(* IEC 61131-3 sources: xPLCCore/codesys_code/Application/APPs, 7 files *)

(* ---- AxisGroupSM.st ---- *)
PROGRAM AxisGroupSM
    VAR CONSTANT
        FlyEventBufferSize: UDINT := 10;
        TaskInstructionBufferSize: UDINT := 10;
        FlyEventStageLimit: INT := 9;

        // Motion buffer fullness threshold: reject new 'M' packets when the
        // SoftMotion command buffer has this many queued moves (back-pressure).
        MOTION_BUFFER_THRESHOLD : ULINT := 12;
        // Cooldown (ms) before re-trying a motion command after the FB
        // refused .CommandAccepted (e.g. GroupWait, MoveLinearAbsolute).
        RETRY_COOLDOWN_G4_MS    : DINT := 100;
        RETRY_COOLDOWN_G1_MS    : DINT := 101;
        // Error code reported on FlyEvent TimeToLive expiry.
        TRIGGER_TIMEOUT_ERR     : INT := 100;
        // Sentinel used by 'G1' to detect "A not supplied" in the TryReadREAL
        // default. Any real A value is << |919191|.
        G1_A_UNSET_SENTINEL     : LREAL := -919191;
    END_VAR
    VAR
        reelpullmotor_fActPosition:REAL;
		OutputCHs:ARRAY[0..15] OF USINT;
		InputCHs:ARRAY[0..15] OF USINT;
		RuntimeMs: LINT := 0;
        BusPeriod: DINT := 1;
        AxisGroupReady: BOOL := FALSE;

        AxisGroupManagerFb: AxisGroupManager(
            agAxisGroup := AxisGroupGVL_agSpiderR.SpiderR,
			axReel:=reelpullmotor);

        GroupActualPositionFb: SM3_Robotics.MC_GroupReadActualPosition;
        ReadPosition: SM3_Robotics.SMC_POS_REF;

        SetCoordTransformFb : MC_SetCoordinateTransform;
        ReadMcsTransformFb : MC_ReadCoordinateTransform;
        ApplyCoordTransform : BOOL := FALSE;
        CoordTransform : MC_COORD_REF;

        InputEvent: E_RobotEvent := E_RobotEvent.EV_NONE;
        PreviousInputEvent: E_RobotEvent := E_RobotEvent.EV_NONE;
        VisuEventControl: INT;
        StateString: STRING;

        MotionStateString: STRING;

        reelMoveRelative : MC_MoveRelative;
        reelMoveRelative2: MC_MoveRelative;   // second instance: SoftMotion forbids >1 movement per FB
        // Request-pattern vars for cyclic reelMoveRelative
        reelGoRequest  : BOOL  := FALSE;
        reelGoRequest2 : BOOL  := FALSE;
        reelGoDistance : LREAL := 0;
        reelGoVelocity : LREAL := 0;
        reelGoAccel    : LREAL := 100;
        reelGoDecel    : LREAL := 100;
        reelGoJerk     : LREAL := 1000;

        MoveLinearAbsoluteFb: SM3_Robotics.MC_MoveLinearAbsolute;
        GroupWaitFb: SM3_Robotics.SMC_GroupWait;

        MotionPose: SM3_Robotics.SMC_POS_REF := ( c := (x := 0.0, y := 0.0, z := 0.0, a := 0.0));

        PacketType: STRING;
        CommandType: STRING;
        CommandId: DINT := 0;
        ShouldReturn: BOOL := FALSE;
        CommandAck: BOOL := FALSE;

        MessageUnpackerFb: FB_MpUnpacker;
        fbPinOpSeqUnpacker: FB_MpUnpacker; // Helper unpacker for pin_op_seq array

        FlyEventBuffer: ARRAY [0..FlyEventBufferSize-1] OF FlyEventData; // event queue for motion-triggered IO
        FlyEventAvailableCount: INT;

        // TaskInstructionBuffer: ARRAY [0..TaskInstructionBufferSize-1] OF TaskInstructionData;
        // TaskInstructionBuffer_ridx:FB_RingBufferIndex(TaskInstructionBufferSize);

        RetryMotionCommandCooldown: DINT := 0;

        LatestFeedRate: LREAL := 10000;
        LatestAcceleration: LREAL := 10000;
        LatestDeceleration: LREAL := 10000;
        LatestJerk: LREAL := 10000;
        LatestFactor: LREAL := 1;

        CornerTransition: REAL := 3;

        GroupReadStatusFb: SM3_Robotics.MC_GroupReadStatus;
        GroupReadPositionFb: SM3_Robotics.SMC_GroupReadPositionInMovement;
        GroupReadPositionFb2: SM3_Robotics.SMC_GroupReadPositionInMovement;

        MotionBufferSize: ULINT;
        CurrentMovementId: SMC_Movement_Id;
        CurrentMovementIdProgress: REAL;

        MessagePackerFb: FB_MpPacker;
        ResponsePacketPointer: POINTER TO MsgPakInfo;

        // MaxVelocity: REAL := 1000;
        // MaxAcceleration: REAL := 4000;
        // MaxJerk: REAL := 4000000;

        DigitalOutputBits: ULINT;
        TmpDigitalOutputBits: ULINT;

        IoTriggerCount: INT := 0;
        IoTriggerResetCount: INT := 0;
        IoTriggerInfoCount: INT := 0;
        IoCommandCount: INT := 0;

        DigitalInputBits_Curr: ULINT := 0;
        DigitalInputBits_Prev: ULINT := 0;
        DigitalInputFlipCounts: ARRAY[0..15] OF UDINT;

        PrevAxisGroupState: INT := -1; // Force initial StateString update

    Index : INT;
    StageLoopIdx : INT;
    PinOpSeqIdx : INT; // Index for iterating through pin_op_seq array

    TempMovementId : SMC_Movement_Id;

    MessageBufferPointer : POINTER TO BYTE;
    AuxCommandBufferPointer : POINTER TO BYTE;

    TriggerActive : BOOL;
    TriggerErrorCode : INT;
    TempByte : BYTE;
    DigitalOutputPointer : POINTER TO BYTE;

        MotionOutputPin: ULINT;
        StagePinState: ULINT;
        StagePinMaskTemp: ULINT;
        StagePinStateTemp: ULINT;
        StageDelayTemp: DINT;

    //LocVar FOR ProcessMotionPacket
    TransitionParameter : ARRAY [0..1] OF LREAL := [0, 0];
    FlyEventTempData : FlyEventData;
    MotionPoseTempReal : REAL;
    PrevMotionStateId : SMC_Movement_Id; // For MotionStateString change detection
    PrevMotionStateProgress : REAL := -1.0; // Force initial update
    G1AbortMode : BOOL; // TRUE = BufferMode.Aborting, interrupts current move

    G4HaltTime: REAL;
    InputPinMask: UINT;
    InputPinGroup: UINT;
    InputPinState: UINT;

    MotionTargetMovementId: SMC_Movement_Id;

    DigitalInputPointer: POINTER TO BYTE;

    DBG_PIN: UINT;

    DBG_BLOCK : BOOL:=TRUE;

    END_VAR
(* =========== IMPLEMENTATION =========== *)

//IMPORTANT:following if TRUE... and if FALSE.... are mandatory, DO not try to remove/optimize it

    //InitRuntime();
    IF TRUE THEN
        IF RuntimeMs = 0 THEN
            FOR Index := 0 TO GVL.reMP_info_ridx.capacity() - 1 DO
                GVL.reMP_info_arr[Index] := MsgPakInfoInit(
                    buff := ADR(GVL.reMP_info_buf[Index]),
                    buffer_size := GVL.reMP_info_buff_SIZE,
                    useLargeElementCountField := TRUE
                );
            END_FOR
        END_IF;
    END_IF;

    // Virtual-motors TTL gate. Derive GVL.bVirtualMotorsMode from
    // GVL.bVirtualMotorsMode_Request (which the operator forces via
    // CODESYS online mode) and a self-expiring timer. Even if the force
    // is left on indefinitely, the derived flag snaps back to FALSE
    // after VIRTUAL_MOTORS_TTL so a forgotten override can't leak into
    // a real-motor session without a cold boot. See GVL.st for docs.
    GVL.fbVirtualMotorsExpire(IN := GVL.bVirtualMotorsMode_Request, PT := GVL.VIRTUAL_MOTORS_TTL);
    GVL.bVirtualMotorsMode := GVL.bVirtualMotorsMode_Request AND NOT GVL.fbVirtualMotorsExpire.Q;

    //UpdateRuntimeAndInputEvent();
    IF TRUE THEN
        RuntimeMs := RuntimeMs + BusPeriod;

        // VisuEventControl=0 is the idle/no-op default so the TCP handler
        // (ProcessSystemPacket below) can own InputEvent without being
        // clobbered by this block on the next cycle. Visualisation buttons
        // should write 1..6 momentarily and reset to 0.
        CASE VisuEventControl OF
            1: InputEvent := E_RobotEvent.EV_POWER_ON;
            2: InputEvent := E_RobotEvent.EV_GROUP_ENABLE;
            3: InputEvent := E_RobotEvent.EV_HOME_GO;
            4: InputEvent := E_RobotEvent.EV_ERROR;
            5: InputEvent := E_RobotEvent.EV_RESET;
            6: InputEvent := E_RobotEvent.EV_HOME_GO_FORCE_SKIP;
        END_CASE;

        IF (PreviousInputEvent <> InputEvent) THEN
            AxisGroupManagerFb.TRANSITION(
                eEvent := InputEvent
            );
        END_IF;

        PreviousInputEvent := InputEvent;
        IF TO_INT(AxisGroupManagerFb._eState) <> PrevAxisGroupState THEN
            StateString := TO_STRING(AxisGroupManagerFb._eState);
            PrevAxisGroupState := TO_INT(AxisGroupManagerFb._eState);
        END_IF;
    END_IF;

    //UpdateAxisGroupState();
    IF TRUE THEN
        AxisGroupManagerFb.Update();

        GroupReadStatusFb(
            AxisGroup := AxisGroupManagerFb._agAxisGroup,
            Enable := 1,
            ActiveMovementId =>
        );

        GroupReadPositionFb(
            AxisGroup := AxisGroupManagerFb._agAxisGroup,
            Enable := TRUE
        );

        GroupActualPositionFb(
            AxisGroup := AxisGroupManagerFb._agAxisGroup,
            Enable := 1,
            CoordSystem := SMC_COORD_SYSTEM.WCS,
            Position => ReadPosition,
        );

    END_IF;

    // Global error supervisor: the per-state checks in AxisGroupManager.Update
    // only watch the power FBs. A move that goes into errorstop (axis fault,
    // bus drop mid-motion, servo trip) surfaces on GroupReadStatusFb.Error /
    // GroupReadPositionFb.Error, and a bus-level fault on
    // IoConfig_Globals.EtherCAT_Master_SoftMotion.xError. Catch those here
    // and drive the FSM to Error -- guarded so we don't loop while already
    // in Error/UnInited. Bus errors take priority so the error source is
    // diagnostic rather than a downstream symptom.
    IF (AxisGroupManagerFb._eState <> E_RobotState.Error
        AND AxisGroupManagerFb._eState <> E_RobotState.UnInited) THEN
        IF IoConfig_Globals.EtherCAT_Master_SoftMotion.xError THEN
            GVL.LastErrorSource := 'Supervisor:EtherCAT_Master';
            GVL.LastErrorID := 0;
            AxisGroupManagerFb.Transition(E_RobotEvent.EV_ERROR);
        ELSIF GroupReadStatusFb.Error THEN
            GVL.LastErrorSource := 'Supervisor:GroupReadStatus';
            GVL.LastErrorID := TO_DWORD(GroupReadStatusFb.ErrorID);
            AxisGroupManagerFb.Transition(E_RobotEvent.EV_ERROR);
        ELSIF GroupReadPositionFb.Error THEN
            GVL.LastErrorSource := 'Supervisor:GroupReadPosition';
            GVL.LastErrorID := TO_DWORD(GroupReadPositionFb.ErrorID);
            AxisGroupManagerFb.Transition(E_RobotEvent.EV_ERROR);
        END_IF;
    END_IF;

    //UpdateMotionProgress();
    IF TRUE THEN
        TempMovementId := GroupReadPositionFb.MovementId;
        // If either MC read FB is in error, don't propagate its outputs -- they
        // may be stale. Freeze buffer size to 0 so ProcessMotionPacket won't
        // treat "buffer has room" as "motion is healthy" and accept a new
        // move on top of an errored group.
        IF GroupReadStatusFb.Error OR GroupReadPositionFb.Error THEN
            MotionBufferSize := 0;
        ELSIF (GroupReadPositionFb.MovementId = 0) THEN
            MotionBufferSize := 0;
            CurrentMovementId := GroupReadStatusFb.LastAcceptedMovementId;
            CurrentMovementIdProgress := 1;
            IF (CurrentMovementId = 0) THEN
                CurrentMovementIdProgress := 0;
            END_IF;
        ELSE
            // Guard against underflow: both are unsigned SMC_Movement_Id.
            // LastAccepted < current shouldn't happen, but could during
            // a reset race. Clamp to 0 rather than wrapping to huge ULINT.
            IF GroupReadStatusFb.LastAcceptedMovementId >= GroupReadPositionFb.MovementId THEN
                MotionBufferSize := GroupReadStatusFb.LastAcceptedMovementId - GroupReadPositionFb.MovementId;
            ELSE
                MotionBufferSize := 0;
            END_IF;

            IF (CurrentMovementId <> GroupReadPositionFb.MovementId) THEN
                CurrentMovementId := GroupReadPositionFb.MovementId;
            END_IF;

            CurrentMovementIdProgress := GroupReadPositionFb.Position;
        END_IF;

        IF (CurrentMovementId <> PrevMotionStateId OR CurrentMovementIdProgress <> PrevMotionStateProgress) THEN
            MotionStateString := CONCAT(
                CONCAT(TO_STRING(CurrentMovementId), ' '),
                TO_STRING(CurrentMovementIdProgress)
            );
            PrevMotionStateId := CurrentMovementId;
            PrevMotionStateProgress := CurrentMovementIdProgress;
        END_IF;

        ShouldReturn := FALSE;
        CommandAck := FALSE;

    END_IF;

    //ReadIncomingPacket();
    IF TRUE THEN
        PacketType := '';
        ResponsePacketPointer := 0;

        IF (GVL.minfo_buf_ridx.size() > 0) THEN
            MessageBufferPointer := ADR(GVL.minfo_buf[GVL.minfo_buf_ridx.getTail()][0]);
            MessageUnpackerFb.Init(ADR(MessageBufferPointer[1]), MessageBufferPointer[0]);
            CommandId := TO_DINT(MessageUnpackerFb.TryReadINT64('id', - 1));
            PacketType := MessageUnpackerFb.TryReadString('type', '');
            CommandType := MessageUnpackerFb.TryReadString('cmd', '');
        END_IF;
    END_IF;

    IF TRUE THEN//ProcessSystemPacket

        IF (PacketType = 'SYS') THEN
            // reMP overflow guard: if the reply ring is full, drop the oldest
            // queued reply to make room. getHead() returning -1 would index
            // reMP_info_arr[-1] and fault the task. See doc/ringbuf-bugs.md #4.
            IF (GVL.reMP_info_ridx.space() = 0) THEN
                GVL.reMP_info_ridx.consumeTail();
                GVL.ReMpDropCount := GVL.ReMpDropCount + 1;
            END_IF;
            ResponsePacketPointer := ADR(GVL.reMP_info_arr[GVL.reMP_info_ridx.getHead()]); // prepare for return data buffer

            MsgPakInfoClear(ResponsePacketPointer^);

            IF (CommandType = 'GA_EV') THEN
                ShouldReturn := TRUE;
                CommandAck := TRUE;
                InputEvent := TO_UDINT(MessageUnpackerFb.TryReadINT64('ev', - 1));
                AxisGroupManagerFb.TRANSITION(
                    eEvent := InputEvent
                );

                ShouldReturn := TRUE;
                CommandAck := TRUE;
                ResponsePacketPointer^.ele_count := 4;
                ResponsePacketPointer^.whead := MessagePackerFb.PackString(pStart := ResponsePacketPointer^.whead, psValue := ADR('st'));
                ResponsePacketPointer^.whead := MessagePackerFb.PackDINT(pStart := ResponsePacketPointer^.whead, diValue := AxisGroupManagerFb._eState);
                ResponsePacketPointer^.whead := MessagePackerFb.PackString(pStart := ResponsePacketPointer^.whead, psValue := ADR('st_str'));
                StateString := TO_STRING(AxisGroupManagerFb._eState);
                PrevAxisGroupState := TO_INT(AxisGroupManagerFb._eState);
                ResponsePacketPointer^.whead := MessagePackerFb.PackString(pStart := ResponsePacketPointer^.whead, psValue := ADR(StateString));
                // Error latch: empty string + 0 when no error has been recorded
                // since the last EV_RESET -> UnInited cycle.
                ResponsePacketPointer^.whead := MessagePackerFb.PackString(pStart := ResponsePacketPointer^.whead, psValue := ADR('err_src'));
                ResponsePacketPointer^.whead := MessagePackerFb.PackString(pStart := ResponsePacketPointer^.whead, psValue := ADR(GVL.LastErrorSource));
                ResponsePacketPointer^.whead := MessagePackerFb.PackString(pStart := ResponsePacketPointer^.whead, psValue := ADR('err_id'));
                ResponsePacketPointer^.whead := MessagePackerFb.PackDINT(pStart := ResponsePacketPointer^.whead, diValue := TO_DINT(GVL.LastErrorID));
            ELSE
                // Unknown SYS command -- emit NAK so the TS caller doesn't hang on timeout.
                ShouldReturn := TRUE;
                CommandAck := FALSE;
                ResponsePacketPointer^.ele_count := 1;
                ResponsePacketPointer^.whead := MessagePackerFb.PackString(pStart := ResponsePacketPointer^.whead, psValue := ADR('err'));
                ResponsePacketPointer^.whead := MessagePackerFb.PackString(pStart := ResponsePacketPointer^.whead, psValue := ADR('unknown SYS cmd'));
            END_IF;

            GVL.minfo_buf_ridx.consumeTail();

            IF ShouldReturn = TRUE THEN // return ack/nak with id
                ResponsePacketPointer^.whead := MessagePackerFb.PackString(pStart := ResponsePacketPointer^.whead, psValue := ADR('id'));
                ResponsePacketPointer^.whead := MessagePackerFb.PackDINT(pStart := ResponsePacketPointer^.whead, diValue := CommandId);

                ResponsePacketPointer^.whead := MessagePackerFb.PackString(pStart := ResponsePacketPointer^.whead, psValue := ADR('ack'));
                ResponsePacketPointer^.whead := MessagePackerFb.PackBool(pStart := ResponsePacketPointer^.whead, bValue := CommandAck);

                ResponsePacketPointer^.ele_count := ResponsePacketPointer^.ele_count + 2;
                MsgPakInfoWrapup(ResponsePacketPointer^);
                GVL.reMP_info_ridx.pushHead();
            END_IF;
        END_IF;

    END_IF;

    IF TRUE THEN//ProcessAuxCommands
        // AUX command threads: currently drained without parsing so their ring
        // buffers don't back up and block the client. Wire a real handler here
        // when the AUX command feature is implemented (see README §P2 #10).
        IF (GVL.aux0_info_buf_ridx.size() > 0) THEN
            AuxCommandBufferPointer := ADR(GVL.aux0_info_buf[GVL.aux0_info_buf_ridx.getTail()][0]);
            GVL.aux0_info_buf_ridx.consumeTail();
        END_IF;

        IF (GVL.aux1_info_buf_ridx.size() > 0) THEN
            AuxCommandBufferPointer := ADR(GVL.aux1_info_buf[GVL.aux1_info_buf_ridx.getTail()][0]);
            GVL.aux1_info_buf_ridx.consumeTail();
        END_IF;

        IF (GVL.aux2_info_buf_ridx.size() > 0) THEN
            AuxCommandBufferPointer := ADR(GVL.aux2_info_buf[GVL.aux2_info_buf_ridx.getTail()][0]);
            GVL.aux2_info_buf_ridx.consumeTail();
        END_IF;
    END_IF;

   //OutputCHs[1]:=InputCHs[1];
   //OutputCHs[2]:=InputCHs[2];
   //OutputCHs[3]:=InputCHs[2];

   // DigitalInputPointer := IoConfig_Globals.HECAT_1616.InputData;//////////////////////////////////////////////

    IF DigitalInputPointer <> 0 THEN//TrackDigitalInputFlips
        DigitalInputBits_Curr := TO_ULINT(DigitalInputPointer[0]) OR SHL(TO_ULINT(DigitalInputPointer[1]), 8);
        IF RuntimeMs > 1 THEN
            TmpDigitalOutputBits := DigitalInputBits_Curr XOR DigitalInputBits_Prev;
            IF TmpDigitalOutputBits <> 0 THEN
                FOR Index := 0 TO 15 DO
                    IF (SHR(TmpDigitalOutputBits, TO_DINT(Index)) AND 1) <> 0 THEN
                        DigitalInputFlipCounts[Index] := DigitalInputFlipCounts[Index] + 1;
                    END_IF;
                END_FOR;
            END_IF;
        END_IF;
        DigitalInputBits_Prev := DigitalInputBits_Curr;
    END_IF;

    IF TRUE THEN//CheckAxisGroupReady
        AxisGroupReady := (AxisGroupManagerFb._eState = E_RobotState.Ready);

        IF NOT AxisGroupReady THEN
            // Host-authority gate (solidification.md W1 A1). Previously this
            // block called GVL.minfo_buf_ridx.clear() which silently dropped
            // every queued motion packet with no reply -- the UI's
            // sendTcpMsgPack would hang until its own timeout. Drain each
            // packet with an explicit NAK + err='group_not_ready' so the
            // host can distinguish "PLC not ready" from "PLC dead".
            // SYS/AUX paths above already ran and are unaffected.
            WHILE GVL.minfo_buf_ridx.size() > 0 DO
                // Re-parse each slot's header to get CommandId for the echo.
                MessageBufferPointer := ADR(GVL.minfo_buf[GVL.minfo_buf_ridx.getTail()][0]);
                MessageUnpackerFb.Init(ADR(MessageBufferPointer[1]), MessageBufferPointer[0]);
                CommandId := TO_DINT(MessageUnpackerFb.TryReadINT64('id', -1));

                // reMP overflow guard (see doc/ringbuf-bugs.md #4).
                IF (GVL.reMP_info_ridx.space() = 0) THEN
                    GVL.reMP_info_ridx.consumeTail();
                    GVL.ReMpDropCount := GVL.ReMpDropCount + 1;
                END_IF;
                ResponsePacketPointer := ADR(GVL.reMP_info_arr[GVL.reMP_info_ridx.getHead()]);
                MsgPakInfoClear(ResponsePacketPointer^);
                ResponsePacketPointer^.ele_count := ResponsePacketPointer^.ele_count + 3;
                ResponsePacketPointer^.whead := MessagePackerFb.PackString(pStart := ResponsePacketPointer^.whead, psValue := ADR('err'));
                ResponsePacketPointer^.whead := MessagePackerFb.PackString(pStart := ResponsePacketPointer^.whead, psValue := ADR('group_not_ready'));
                ResponsePacketPointer^.whead := MessagePackerFb.PackString(pStart := ResponsePacketPointer^.whead, psValue := ADR('id'));
                ResponsePacketPointer^.whead := MessagePackerFb.PackDINT(pStart := ResponsePacketPointer^.whead, diValue := CommandId);
                ResponsePacketPointer^.whead := MessagePackerFb.PackString(pStart := ResponsePacketPointer^.whead, psValue := ADR('ack'));
                ResponsePacketPointer^.whead := MessagePackerFb.PackBool(pStart := ResponsePacketPointer^.whead, bValue := FALSE);
                MsgPakInfoWrapup(ResponsePacketPointer^);
                GVL.reMP_info_ridx.pushHead();

                GVL.minfo_buf_ridx.consumeTail();
                GVL.GroupNotReadyNakCount := GVL.GroupNotReadyNakCount + 1;
            END_WHILE;

            MotionPose.c.X := 0;
            MotionPose.c.Y := 0;
            MotionPose.c.Z := 0;
            MotionPose.c.A := 0;
            MotionPose.c.B := 0;
            MotionPose.c.C := 0;
        END_IF;
    END_IF;

    IF NOT AxisGroupReady THEN
        RETURN;
    END_IF;

    IF FALSE THEN///ProcessTaskPacket

        IF (PacketType = 'TASK') THEN
            ResponsePacketPointer := ADR(GVL.reMP_info_arr[GVL.reMP_info_ridx.getHead()]); // prepare for return data buffer

            MsgPakInfoClear(ResponsePacketPointer^);

            IF (CommandType = 'GA_EV') THEN
            	Index:=0;
            END_IF;

            GVL.minfo_buf_ridx.consumeTail();

            IF ShouldReturn = TRUE THEN // return ack/nak with id
                ResponsePacketPointer^.whead := MessagePackerFb.PackString(pStart := ResponsePacketPointer^.whead, psValue := ADR('id'));
                ResponsePacketPointer^.whead := MessagePackerFb.PackDINT(pStart := ResponsePacketPointer^.whead, diValue := CommandId);

                ResponsePacketPointer^.whead := MessagePackerFb.PackString(pStart := ResponsePacketPointer^.whead, psValue := ADR('ack'));
                ResponsePacketPointer^.whead := MessagePackerFb.PackBool(pStart := ResponsePacketPointer^.whead, bValue := CommandAck);

                ResponsePacketPointer^.ele_count := ResponsePacketPointer^.ele_count + 2;
                MsgPakInfoWrapup(ResponsePacketPointer^);
                GVL.reMP_info_ridx.pushHead();
            END_IF;
        END_IF;

    END_IF;

    IF TRUE THEN//ProcessFlyEventsAndIo

        TriggerActive := FALSE;
        FlyEventAvailableCount := 0;

        FOR Index := 0 TO TO_INT(FlyEventBufferSize - 1) DO
            TriggerActive := FALSE;
            TriggerErrorCode := 0;

            CASE FlyEventBuffer[Index].TriggerType OF
                FlyEventTriggerType.MovmentProgressTrigger:
                    IF (
                        CurrentMovementId > FlyEventBuffer[Index].TargetMovementId OR
                        (CurrentMovementId = FlyEventBuffer[Index].TargetMovementId AND CurrentMovementIdProgress >= FlyEventBuffer[Index].TargetMovementProgress)
                    ) THEN
                        TriggerActive := TRUE;
                        IF (FlyEventBuffer[Index].IoStageCount > 0) THEN
                            FlyEventBuffer[Index].IoStageIndex := 0;
                            FlyEventBuffer[Index].IoStageDelayCountdown := FlyEventBuffer[Index].IoStageDelay[0];
                            FlyEventBuffer[Index].TriggerType := FlyEventTriggerType.SequenceDelayWait;
                            IF (FlyEventBuffer[Index].IoStageDelayCountdown > 0) THEN
                                TriggerActive := FALSE;
                            END_IF;
                        END_IF;
                    ELSE
                        IF (FlyEventBuffer[Index].TimeToLiveMs > 0) THEN
                            FlyEventBuffer[Index].TimeToLiveMs := FlyEventBuffer[Index].TimeToLiveMs - BusPeriod;
                            IF (FlyEventBuffer[Index].TimeToLiveMs <= 0) THEN
                                TriggerActive := TRUE;
                                TriggerErrorCode := TRIGGER_TIMEOUT_ERR;
                            END_IF;
                        END_IF;
                    END_IF;

                FlyEventTriggerType.SequenceDelayWait:
                    IF (FlyEventBuffer[Index].IoStageIndex < FlyEventBuffer[Index].IoStageCount) THEN
                        FlyEventBuffer[Index].IoStageDelayCountdown := FlyEventBuffer[Index].IoStageDelayCountdown - BusPeriod;
                        IF (FlyEventBuffer[Index].IoStageDelayCountdown <= 0) THEN
                            TriggerActive := TRUE;
                        END_IF;
                    END_IF;

                FlyEventTriggerType.NOP:
                    FlyEventAvailableCount := FlyEventAvailableCount + 1;
            END_CASE;

            IF (TriggerActive = FALSE) THEN
                CONTINUE;
            END_IF;

            IF (TriggerErrorCode <> 0) THEN
                // reMP overflow guard (see doc/ringbuf-bugs.md #4).
                IF (GVL.reMP_info_ridx.space() = 0) THEN
                    GVL.reMP_info_ridx.consumeTail();
                    GVL.ReMpDropCount := GVL.ReMpDropCount + 1;
                END_IF;
                ResponsePacketPointer := ADR(GVL.reMP_info_arr[GVL.reMP_info_ridx.getHead()]); // prepare for return data buffer
                MsgPakInfoClear(ResponsePacketPointer^);
                ResponsePacketPointer^.ele_count := ResponsePacketPointer^.ele_count + 3;

                ResponsePacketPointer^.whead := MessagePackerFb.PackString(pStart := ResponsePacketPointer^.whead, psValue := ADR('error_code'));
                ResponsePacketPointer^.whead := MessagePackerFb.PackDINT(pStart := ResponsePacketPointer^.whead, diValue := TriggerErrorCode);

                ResponsePacketPointer^.whead := MessagePackerFb.PackString(pStart := ResponsePacketPointer^.whead, psValue := ADR('src_id'));
                ResponsePacketPointer^.whead := MessagePackerFb.PackDINT(pStart := ResponsePacketPointer^.whead, diValue := FlyEventBuffer[Index].SourceCommandId);

                ResponsePacketPointer^.whead := MessagePackerFb.PackString(pStart := ResponsePacketPointer^.whead, psValue := ADR('event_id'));
                ResponsePacketPointer^.whead := MessagePackerFb.PackLINT(pStart := ResponsePacketPointer^.whead, liValue := TO_LINT(FlyEventBuffer[Index].EventId));

                MsgPakInfoWrapup(ResponsePacketPointer^);
                GVL.reMP_info_ridx.pushHead();

                FlyEventBuffer[Index].ActionType := FlyEventActType.NOP;
                FlyEventBuffer[Index].TriggerType := FlyEventTriggerType.NOP;
            ELSE
                CASE FlyEventBuffer[Index].ActionType OF
                    FlyEventActType.PIN_OPERATION:
                        IF (FlyEventBuffer[Index].IoStageCount > 0) THEN
                            MotionOutputPin := FlyEventBuffer[Index].IoStagePinMask[FlyEventBuffer[Index].IoStageIndex];
                            StagePinState := FlyEventBuffer[Index].IoStagePinState[FlyEventBuffer[Index].IoStageIndex];
                        ELSE
                            MotionOutputPin := 0;
                            StagePinState := 0;
                        END_IF;

                        TmpDigitalOutputBits := DigitalOutputBits;
                        TmpDigitalOutputBits :=
                            (TmpDigitalOutputBits AND NOT (MotionOutputPin)) OR
                            ((StagePinState) AND (MotionOutputPin));
                        DigitalOutputBits := TmpDigitalOutputBits;

                        FlyEventBuffer[Index].IoStageIndex := FlyEventBuffer[Index].IoStageIndex + 1;
                        IF (FlyEventBuffer[Index].IoStageIndex < FlyEventBuffer[Index].IoStageCount) THEN
                            FlyEventBuffer[Index].IoStageDelayCountdown := FlyEventBuffer[Index].IoStageDelay[FlyEventBuffer[Index].IoStageIndex];
                            FlyEventBuffer[Index].TriggerType := FlyEventTriggerType.SequenceDelayWait;
                        ELSE
                            FlyEventBuffer[Index].ActionType := FlyEventActType.NOP;
                            FlyEventBuffer[Index].TriggerType := FlyEventTriggerType.NOP;
                        END_IF;

                        IoTriggerCount := IoTriggerCount + 1;

                    FlyEventActType.ACK_SRC_ID://send ack with source command id
                        // reMP overflow guard (see doc/ringbuf-bugs.md #4).
                        IF (GVL.reMP_info_ridx.space() = 0) THEN
                            GVL.reMP_info_ridx.consumeTail();
                            GVL.ReMpDropCount := GVL.ReMpDropCount + 1;
                        END_IF;

                        ResponsePacketPointer := ADR(GVL.reMP_info_arr[GVL.reMP_info_ridx.getHead()]); // prepare for return data buffer
                        MsgPakInfoClear(ResponsePacketPointer^);

                        ResponsePacketPointer^.ele_count := ResponsePacketPointer^.ele_count +3;//three elements: event_id, id, ack

                        ResponsePacketPointer^.whead := MessagePackerFb.PackString(pStart := ResponsePacketPointer^.whead, psValue := ADR('event_id'));
                        ResponsePacketPointer^.whead := MessagePackerFb.PackLINT(pStart := ResponsePacketPointer^.whead, liValue := TO_LINT(FlyEventBuffer[Index].EventId));

                        ResponsePacketPointer^.whead := MessagePackerFb.PackString(pStart := ResponsePacketPointer^.whead, psValue := ADR('id'));
                        ResponsePacketPointer^.whead := MessagePackerFb.PackDINT(pStart := ResponsePacketPointer^.whead, diValue := FlyEventBuffer[Index].SourceCommandId);

                        ResponsePacketPointer^.whead := MessagePackerFb.PackString(pStart := ResponsePacketPointer^.whead, psValue := ADR('ack'));
                        ResponsePacketPointer^.whead := MessagePackerFb.PackBool(pStart := ResponsePacketPointer^.whead, bValue := TRUE);

                        MsgPakInfoWrapup(ResponsePacketPointer^);
                        GVL.reMP_info_ridx.pushHead();

                        // IF (FlyEventBuffer[Index].SourceCommandId = CommandId) THEN
                        //     TriggerActive := TRUE;
                        // END_IF;

                        FlyEventBuffer[Index].ActionType := FlyEventActType.NOP;
                        FlyEventBuffer[Index].TriggerType := FlyEventTriggerType.NOP;

                END_CASE;
            END_IF;

            IoTriggerInfoCount := IoTriggerInfoCount + 1;
        END_FOR;

        //DigitalOutputPointer := IoConfig_Globals.HECAT_1616.OutputData;//////////////////////////////////////////////
        OutputCHs[0] := TO_BYTE(DigitalOutputBits AND 16#FF);
        OutputCHs[1] := TO_BYTE(SHR(DigitalOutputBits,8) AND 16#FF);

		DBG_PIN:=0;
		IF((DigitalOutputBits AND 16#4000)  >0)THEN
			DBG_PIN:=1;
		END_IF
        MoveLinearAbsoluteFb(
            AxisGroup := AxisGroupManagerFb._agAxisGroup,
            Execute := 0
        );

        GroupWaitFb(
            AxisGroup := AxisGroupManagerFb._agAxisGroup,
            Execute := 0
        );

        IF (RetryMotionCommandCooldown > 0) THEN
            RetryMotionCommandCooldown := RetryMotionCommandCooldown - BusPeriod;
        END_IF;

        SetCoordTransformFb(
            AxisGroup := AxisGroupManagerFb._agAxisGroup,
            Execute := ApplyCoordTransform,
            CoordTransform := CoordTransform,
            CoordSystem := SMC_COORD_SYSTEM.MCS
        );

        IF ApplyCoordTransform AND (SetCoordTransformFb.Busy OR SetCoordTransformFb.Done OR SetCoordTransformFb.Error) THEN
            ApplyCoordTransform := FALSE;
        END_IF;

        ReadMcsTransformFb(
            AxisGroup := AxisGroupManagerFb._agAxisGroup,
            Enable := TRUE,
            CoordSystem := SMC_COORD_SYSTEM.MCS,
            Valid => ,
            Busy => ,
            Error => ,
            ErrorID => ,
            CoordTransform =>
        );
    END_IF;

    reelpullmotor_fActPosition:=reelpullmotor.fActPosition;

    IF TRUE THEN//ProcessMotionPacket

        IF (RetryMotionCommandCooldown = 0 AND PacketType = 'M' AND GVL.minfo_buf_ridx.size() > 0 AND MotionBufferSize < MOTION_BUFFER_THRESHOLD) THEN
            ShouldReturn := FALSE;
            CommandAck := FALSE;

            // reMP overflow guard (see doc/ringbuf-bugs.md #4).
            IF (GVL.reMP_info_ridx.space() = 0) THEN
                GVL.reMP_info_ridx.consumeTail();
                GVL.ReMpDropCount := GVL.ReMpDropCount + 1;
            END_IF;
            ResponsePacketPointer := ADR(GVL.reMP_info_arr[GVL.reMP_info_ridx.getHead()]); // prepare for return data buffer
            MsgPakInfoClear(ResponsePacketPointer^);

            IF (GroupReadStatusFb.Error = TRUE OR GroupReadStatusFb.GroupErrorStop) THEN
                ResponsePacketPointer^.ele_count := ResponsePacketPointer^.ele_count + 1;
                ResponsePacketPointer^.whead := MessagePackerFb.PackString(pStart := ResponsePacketPointer^.whead, psValue := ADR('ERROR_CODE'));
                ResponsePacketPointer^.whead := MessagePackerFb.PackLINT(pStart := ResponsePacketPointer^.whead, liValue := GroupReadStatusFb.ErrorID);

                IF (GroupReadStatusFb.GroupErrorStop) THEN
                    ResponsePacketPointer^.ele_count := ResponsePacketPointer^.ele_count + 1;
                    ResponsePacketPointer^.whead := MessagePackerFb.PackString(pStart := ResponsePacketPointer^.whead, psValue := ADR('MISC'));
                    ResponsePacketPointer^.whead := MessagePackerFb.PackString(pStart := ResponsePacketPointer^.whead, psValue := ADR('GroupErrorStop'));
                END_IF;

                ShouldReturn := TRUE;
                CommandAck := FALSE;
                GVL.minfo_buf_ridx.consumeTail();

            ELSIF (CommandType = 'BLOCK_FOR_MOTION_STOP') THEN
                IF (GroupReadPositionFb.MovementId = 0) THEN
                    ShouldReturn := TRUE;
                    CommandAck := TRUE;

                    GVL.minfo_buf_ridx.consumeTail();
                END_IF;

            ELSIF (CommandType = 'BLOCK_FOR_DIGITAL_INPUT') THEN
                InputPinMask := TO_UINT(MessageUnpackerFb.TryReadINT64('pin', 0));
                InputPinGroup := TO_UINT(MessageUnpackerFb.TryReadINT64('group', 0));
                InputPinState := TO_UINT(MessageUnpackerFb.TryReadINT64('state', 0));

                IF DigitalInputPointer <> 0 AND ((DigitalInputPointer[InputPinGroup] AND InputPinMask) = (InputPinState AND InputPinMask)) THEN
                    ShouldReturn := TRUE;
                    CommandAck := TRUE;

                    GVL.minfo_buf_ridx.consumeTail();
                END_IF;
            ELSIF (CommandType = 'GET_DIGITAL_INPUT') THEN
                //InputPinGroup := TO_UINT(MessageUnpackerFb.TryReadINT64('group', 0));

                ResponsePacketPointer^.ele_count := ResponsePacketPointer^.ele_count + 1;

                ResponsePacketPointer^.whead := MessagePackerFb.PackString(pStart := ResponsePacketPointer^.whead, psValue := ADR('state'));
                IF DigitalInputPointer <> 0 THEN
                    ResponsePacketPointer^.whead := MessagePackerFb.PackDINT(pStart := ResponsePacketPointer^.whead,diValue:=DigitalInputPointer[0]OR  SHL( TO_UDINT( DigitalInputPointer[1]),8));
                ELSE
                    // DigitalInputPointer not wired (HECAT_1616 line in TrackDigitalInputFlips is commented out).
                    // Return 0 rather than dereferencing null.
                    ResponsePacketPointer^.whead := MessagePackerFb.PackDINT(pStart := ResponsePacketPointer^.whead, diValue := 0);
                END_IF;

                ShouldReturn := TRUE;
                CommandAck := TRUE;
                GVL.minfo_buf_ridx.consumeTail();
            ELSIF (CommandType = 'READ_LATEST_CMD_LOCATION') THEN
                ResponsePacketPointer^.ele_count := ResponsePacketPointer^.ele_count + 6;

                ResponsePacketPointer^.whead := MessagePackerFb.PackString(pStart := ResponsePacketPointer^.whead, psValue := ADR('X'));
                ResponsePacketPointer^.whead := MessagePackerFb.PackREAL(pStart := ResponsePacketPointer^.whead, rValue := TO_REAL(MotionPose.c.X));
                ResponsePacketPointer^.whead := MessagePackerFb.PackString(pStart := ResponsePacketPointer^.whead, psValue := ADR('Y'));
                ResponsePacketPointer^.whead := MessagePackerFb.PackREAL(pStart := ResponsePacketPointer^.whead, rValue := TO_REAL(MotionPose.c.Y));
                ResponsePacketPointer^.whead := MessagePackerFb.PackString(pStart := ResponsePacketPointer^.whead, psValue := ADR('Z'));
                ResponsePacketPointer^.whead := MessagePackerFb.PackREAL(pStart := ResponsePacketPointer^.whead, rValue := TO_REAL(MotionPose.c.Z));
                ResponsePacketPointer^.whead := MessagePackerFb.PackString(pStart := ResponsePacketPointer^.whead, psValue := ADR('A'));
                ResponsePacketPointer^.whead := MessagePackerFb.PackREAL(pStart := ResponsePacketPointer^.whead, rValue := TO_REAL(MotionPose.c.A));
                ResponsePacketPointer^.whead := MessagePackerFb.PackString(pStart := ResponsePacketPointer^.whead, psValue := ADR('B'));
                ResponsePacketPointer^.whead := MessagePackerFb.PackREAL(pStart := ResponsePacketPointer^.whead, rValue := TO_REAL(MotionPose.c.B));
                ResponsePacketPointer^.whead := MessagePackerFb.PackString(pStart := ResponsePacketPointer^.whead, psValue := ADR('C'));
                ResponsePacketPointer^.whead := MessagePackerFb.PackREAL(pStart := ResponsePacketPointer^.whead, rValue := TO_REAL(MotionPose.c.C));

                ShouldReturn := TRUE;
                CommandAck := TRUE;
                GVL.minfo_buf_ridx.consumeTail();

            ELSIF (CommandType = 'G4') THEN
                ShouldReturn := TRUE;
                CommandAck := TRUE;
                G4HaltTime := MessageUnpackerFb.TryReadREAL('P', - 1);

                IF (G4HaltTime > 0) THEN
                    GroupWaitFb(
                        AxisGroup := AxisGroupManagerFb._agAxisGroup,
                        Execute := 1,
                        WaitTime := G4HaltTime
                    );

                    IF (GroupWaitFb.CommandAccepted) THEN
                        GVL.minfo_buf_ridx.consumeTail();
                        ResponsePacketPointer^.ele_count := ResponsePacketPointer^.ele_count + 1;

                        ResponsePacketPointer^.whead := MessagePackerFb.PackString(pStart := ResponsePacketPointer^.whead, psValue := ADR('movement_id'));
                        ResponsePacketPointer^.whead := MessagePackerFb.PackLINT(pStart := ResponsePacketPointer^.whead, liValue := TO_LINT(GroupWaitFb.MovementId));

                        ShouldReturn := TRUE;
                        CommandAck := TRUE;
                    ELSE
                        RetryMotionCommandCooldown := RETRY_COOLDOWN_G4_MS;
                    END_IF;
                ELSE
                    GVL.minfo_buf_ridx.consumeTail();

                    ShouldReturn := TRUE;
                    CommandAck := FALSE;
                END_IF;

            ELSIF (CommandType = 'SetCoord0') THEN
                CoordTransform.X := 0.0;
                CoordTransform.Y := 0.0;
                CoordTransform.Z := 0.0;
                CoordTransform.A := 0.0;
                CoordTransform.B := 0.0;
                CoordTransform.C := 0.0;
                ApplyCoordTransform := TRUE;

                ShouldReturn := TRUE;
                CommandAck := TRUE;
                GVL.minfo_buf_ridx.consumeTail();

            ELSIF (CommandType = 'SetCoord1') THEN
                CoordTransform.X := 0.0;
                CoordTransform.Y := 0.0;
                CoordTransform.Z := 0.0;
                CoordTransform.A := 60.0;
                CoordTransform.B := 0.0;
                CoordTransform.C := 0.0;
                ApplyCoordTransform := TRUE;

                ShouldReturn := TRUE;
                CommandAck := TRUE;
                GVL.minfo_buf_ridx.consumeTail();

            ELSIF (CommandType = 'RESET_DBG_INFO') THEN
                IoTriggerCount := 0;
                IoTriggerResetCount := 0;
                IoTriggerInfoCount := 0;
                IoCommandCount := 0;

                ShouldReturn := TRUE;
                CommandAck := TRUE;
                GVL.minfo_buf_ridx.consumeTail();

            ELSIF (CommandType = 'ReelGo') THEN
                reelGoDistance := MessageUnpackerFb.TryReadREAL('Distance', reelGoDistance);
                reelGoVelocity := MessageUnpackerFb.TryReadREAL('F',        reelGoVelocity);
                reelGoAccel    := MessageUnpackerFb.TryReadREAL('ACC',      reelGoAccel);
                reelGoDecel    := MessageUnpackerFb.TryReadREAL('DEA',      reelGoDecel);
                reelGoJerk     := MessageUnpackerFb.TryReadREAL('JERK',     reelGoJerk);

                // Dispatch to whichever FB instance is not currently busy.
                // If both are busy (active + queued), drop the command.
                IF NOT reelMoveRelative.Busy THEN
                    reelGoRequest  := TRUE;
                ELSIF NOT reelMoveRelative2.Busy THEN
                    reelGoRequest2 := TRUE;
                END_IF;

                ShouldReturn := TRUE;
                CommandAck := TRUE;
                GVL.minfo_buf_ridx.consumeTail();

            ELSIF (CommandType = 'M4') THEN

				MotionTargetMovementId := TO_ULINT(MessageUnpackerFb.TryReadUINT64('motion_id', TO_ULINT(GroupReadStatusFb.LastAcceptedMovementId)));

				ResponsePacketPointer^.ele_count := ResponsePacketPointer^.ele_count + 1;

				ResponsePacketPointer^.whead := MessagePackerFb.PackString(pStart := ResponsePacketPointer^.whead, psValue := ADR('ev_buf_space'));

				ResponsePacketPointer^.whead := MessagePackerFb.PackLINT(pStart := ResponsePacketPointer^.whead, liValue := TO_LINT(FlyEventAvailableCount));

				IF (FlyEventAvailableCount > 3) THEN

					FlyEventTempData.ActionType := FlyEventActType.PIN_OPERATION;

					FlyEventTempData.TriggerType := FlyEventTriggerType.MovmentProgressTrigger;

					FlyEventTempData.SourceCommandId := CommandId;

					FlyEventTempData.PinGrp := 0;

					FlyEventTempData.ResetDelayMs := TO_INT(MessageUnpackerFb.TryReadINT64('reset_ms', 0));

					FlyEventTempData.TimeToLiveMs := TO_DINT(MessageUnpackerFb.TryReadINT64('ttl_ms', -1));

					FlyEventTempData.TargetMovementId := MotionTargetMovementId + TO_INT(MessageUnpackerFb.TryReadINT64('motion_id_offset', 0));

					FlyEventTempData.TargetMovementProgress := TO_LREAL(MessageUnpackerFb.TryReadREAL('motion_progress', 1));

					FlyEventTempData.EventId := TO_DINT(MessageUnpackerFb.TryReadINT64('event_id', 0));

					FlyEventTempData.IoStageCount := 0;

					FlyEventTempData.IoStageIndex := 0;

					FlyEventTempData.IoStageDelayCountdown := 0;

					FOR StageLoopIdx := 0 TO FlyEventStageLimit-1 DO

						FlyEventTempData.IoStageDelay[StageLoopIdx] := 0;

						FlyEventTempData.IoStagePinMask[StageLoopIdx] := 0;

						FlyEventTempData.IoStagePinState[StageLoopIdx] := 0;

					END_FOR;

					(* Parse pin_op_seq array: [delay0, pin0, state0, delay1, pin1, state1, ...] *)
					(* Use sequential reading with array unpacker for fast performance - no string operations *)
					IF MessageUnpackerFb.TryReadObject('pin_op_seq', ADR(fbPinOpSeqUnpacker)) THEN
						(* Read array header to get length *)
						fbPinOpSeqUnpacker.UnpackNext();

						(* Loop through array in groups of 3 (delay, pin, state) *)
						FOR PinOpSeqIdx := 0 TO (fbPinOpSeqUnpacker.uiLastCount / 3) - 1 DO
							IF FlyEventTempData.IoStageCount >= FlyEventStageLimit THEN
								EXIT; (* Reached maximum stage limit *)
							END_IF;

							(* Read delay value (signed integer) - sequential read *)
							fbPinOpSeqUnpacker.UnpackNext();
							StageDelayTemp := TO_INT(fbPinOpSeqUnpacker.diLastDINT);

							(* Read pin mask value (unsigned integer) - sequential read *)
							(* UnpackNext reads integers into diLastDINT; convert to ULINT for unsigned values *)
							fbPinOpSeqUnpacker.UnpackNext();
							(* Pin masks are bit patterns, inherently non-negative. Clamp negative
							   DINT values (e.g. client sent a signed negative int by mistake) to 0
							   so we don't wrap into a huge ULINT and trigger unintended outputs. *)
							IF fbPinOpSeqUnpacker.diLastDINT < 0 THEN
								StagePinMaskTemp := 0;
							ELSE
								StagePinMaskTemp := DINT_TO_ULINT(fbPinOpSeqUnpacker.diLastDINT);
							END_IF;

							(* Read pin state value (unsigned integer) - sequential read *)
							fbPinOpSeqUnpacker.UnpackNext();
							IF fbPinOpSeqUnpacker.diLastDINT < 0 THEN
								StagePinStateTemp := 0;
							ELSE
								StagePinStateTemp := DINT_TO_ULINT(fbPinOpSeqUnpacker.diLastDINT);
							END_IF;

							(* Only add stage if pin mask is non-zero *)
							IF StagePinMaskTemp <> 0 THEN
								FlyEventTempData.IoStageDelay[FlyEventTempData.IoStageCount] := StageDelayTemp;
								FlyEventTempData.IoStagePinMask[FlyEventTempData.IoStageCount] := StagePinMaskTemp;
								FlyEventTempData.IoStagePinState[FlyEventTempData.IoStageCount] := StagePinStateTemp;
								FlyEventTempData.IoStageCount := FlyEventTempData.IoStageCount + 1;
							END_IF;
						END_FOR;
					END_IF;

					StagePinMaskTemp := MessageUnpackerFb.TryReadUINT64('pin', 0);

					IF (StagePinMaskTemp <> 0 AND FlyEventTempData.IoStageCount < FlyEventStageLimit) THEN

						StagePinStateTemp := MessageUnpackerFb.TryReadUINT64('state', 0);

						StageDelayTemp := 0;

						FlyEventTempData.IoStageDelay[FlyEventTempData.IoStageCount] := StageDelayTemp;

						FlyEventTempData.IoStagePinMask[FlyEventTempData.IoStageCount] := StagePinMaskTemp;

						FlyEventTempData.IoStagePinState[FlyEventTempData.IoStageCount] := StagePinStateTemp;

						FlyEventTempData.IoStageCount := FlyEventTempData.IoStageCount + 1;

						IF (FlyEventTempData.ResetDelayMs > 0 AND FlyEventTempData.IoStageCount < FlyEventStageLimit) THEN

							FlyEventTempData.IoStageDelay[FlyEventTempData.IoStageCount] := FlyEventTempData.ResetDelayMs;

							FlyEventTempData.IoStagePinMask[FlyEventTempData.IoStageCount] := FlyEventTempData.IoStagePinMask[FlyEventTempData.IoStageCount - 1];

							FlyEventTempData.IoStagePinState[FlyEventTempData.IoStageCount] := ((NOT StagePinStateTemp) AND StagePinMaskTemp);

							FlyEventTempData.IoStageCount := FlyEventTempData.IoStageCount + 1;

						END_IF;

					END_IF;

					IF (FlyEventTempData.IoStageCount > 0 AND MotionTargetMovementId <> 0) THEN

						FOR Index := 0 TO TO_INT( FlyEventBufferSize - 1) DO

							IF (FlyEventBuffer[Index].TriggerType = 0) THEN

								FlyEventBuffer[Index] := FlyEventTempData;

								CommandAck := TRUE;

								EXIT;

							END_IF;

						END_FOR;

						IoCommandCount := IoCommandCount + 1;

						ShouldReturn := TRUE;

					END_IF;

					GVL.minfo_buf_ridx.consumeTail();

				END_IF;

ELSIF (CommandType = 'WAIT_FOR_TRIGGER_MOTION_PROGRESS') THEN
                IF (FlyEventAvailableCount > 3) THEN

                    MotionTargetMovementId := TO_ULINT(MessageUnpackerFb.TryReadINT64('motion_id', TO_LINT(GroupReadStatusFb.LastAcceptedMovementId)));

                    IF (MotionOutputPin <> 0 AND MotionTargetMovementId <> 0) THEN
                        FlyEventTempData.ActionType := FlyEventActType.ACK_SRC_ID;
                        FlyEventTempData.TriggerType := FlyEventTriggerType.MovmentProgressTrigger;
                        FlyEventTempData.TargetMovementId := MotionTargetMovementId + TO_INT(MessageUnpackerFb.TryReadINT64('motion_id_offset', 0));
                        FlyEventTempData.TargetMovementProgress := TO_LREAL(MessageUnpackerFb.TryReadREAL('motion_progress', 1));

                        FlyEventTempData.SourceCommandId := CommandId;

                        FlyEventTempData.EventId := TO_DINT(MessageUnpackerFb.TryReadINT64('event_id', 0));
                        FlyEventTempData.TimeToLiveMs := TO_DINT(MessageUnpackerFb.TryReadINT64('ttl_ms', -1));

                        FOR Index := 0 TO TO_INT(FlyEventBufferSize - 1) DO
                            IF (FlyEventBuffer[Index].TriggerType = 0) THEN
                                FlyEventBuffer[Index] := FlyEventTempData;
                                EXIT;
                            END_IF;
                        END_FOR;
                    END_IF;
                    GVL.minfo_buf_ridx.consumeTail();
                END_IF;

            ELSIF (CommandType = 'G1') THEN
                MotionPose.c.X := MessageUnpackerFb.TryReadREAL('X', MotionPose.c.X);
                MotionPose.c.Y := MessageUnpackerFb.TryReadREAL('Y', MotionPose.c.Y);
                MotionPose.c.Z := MessageUnpackerFb.TryReadREAL('Z', MotionPose.c.Z);
                MotionPoseTempReal := MessageUnpackerFb.TryReadREAL('A', G1_A_UNSET_SENTINEL);
                IF (MotionPoseTempReal <> G1_A_UNSET_SENTINEL) THEN
                    MotionPose.c.A := MotionPoseTempReal / 10;
                END_IF;

                LatestFeedRate := MessageUnpackerFb.TryReadREAL('F', LatestFeedRate);
                LatestAcceleration := MessageUnpackerFb.TryReadREAL('ACC', LatestAcceleration);
                LatestDeceleration := MessageUnpackerFb.TryReadREAL('DEA', LatestDeceleration);
                LatestJerk := MessageUnpackerFb.TryReadREAL('JERK', LatestJerk);
                LatestFactor := MessageUnpackerFb.TryReadREAL('FAC', LatestFactor);
                IF (LatestFactor > 1) THEN LatestFactor := 1; END_IF;
                IF (LatestFactor < 0.001) THEN LatestFactor := 0.001; END_IF;

                CornerTransition := MessageUnpackerFb.TryReadREAL('Cor', CornerTransition);
                TransitionParameter[0] := CornerTransition;
                G1AbortMode := MessageUnpackerFb.TryReadBool('abort', FALSE);

                MoveLinearAbsoluteFb(
                    AxisGroup := AxisGroupManagerFb._agAxisGroup,
                    Execute := 1,
                    Position := MotionPose,
                    Velocity := LatestFeedRate,
                    Acceleration := LatestAcceleration,
                    Deceleration := LatestDeceleration,
                    Jerk := LatestJerk,
                    CoordSystem := SMC_COORD_SYSTEM.WCS,
                    BufferMode := SEL(G1AbortMode,
                        SEL(CornerTransition >= 1, SM3_Common.MC_BUFFER_MODE.Buffered, SM3_Common.MC_BUFFER_MODE.BlendingNext),
                        SM3_Common.MC_BUFFER_MODE.Aborting),
                    TransitionMode := SM3_Robotics.MC_TRANSITION_MODE.TMCornerDistance,
                    TransitionParameter := TransitionParameter,
                    VelFactor := LatestFactor,
                    AccFactor := LatestFactor,
                    JerkFactor := LatestFactor,
                    TorqueFactor := 1,
                    Done => ,
                    Busy => ,
                    Active => ,
                    MovementId =>
                );

                IF (MoveLinearAbsoluteFb.CommandAccepted) THEN
                    GVL.minfo_buf_ridx.consumeTail();

                    ResponsePacketPointer^.ele_count := ResponsePacketPointer^.ele_count + 1;
                    ResponsePacketPointer^.whead := MessagePackerFb.PackString(pStart := ResponsePacketPointer^.whead, psValue := ADR('movement_id'));
                    ResponsePacketPointer^.whead := MessagePackerFb.PackLINT(pStart := ResponsePacketPointer^.whead, liValue := TO_LINT(MoveLinearAbsoluteFb.MovementId));

                    ShouldReturn := TRUE;
                    CommandAck := TRUE;
                ELSE
                    RetryMotionCommandCooldown := RETRY_COOLDOWN_G1_MS;
                END_IF;

            ELSIF (CommandType = 'getDigitalInputFlipCount') THEN
                ResponsePacketPointer^.ele_count := ResponsePacketPointer^.ele_count + 2; // raw + fc

                ResponsePacketPointer^.whead := MessagePackerFb.PackString(pStart := ResponsePacketPointer^.whead, psValue := ADR('raw'));
                ResponsePacketPointer^.whead := MessagePackerFb.PackDINT(pStart := ResponsePacketPointer^.whead, diValue := TO_DINT(DigitalInputBits_Curr));

                ResponsePacketPointer^.whead := MessagePackerFb.PackString(pStart := ResponsePacketPointer^.whead, psValue := ADR('fc'));
                ResponsePacketPointer^.whead := MessagePackerFb.PackArrayHeader(pStart := ResponsePacketPointer^.whead, uiCount := 16);
                FOR StageLoopIdx := 0 TO 15 DO
                    ResponsePacketPointer^.whead := MessagePackerFb.PackDINT(pStart := ResponsePacketPointer^.whead, diValue := TO_DINT(DigitalInputFlipCounts[StageLoopIdx]));
                END_FOR;

                ShouldReturn := TRUE;
                CommandAck := TRUE;
                GVL.minfo_buf_ridx.consumeTail();

            ELSE
                GVL.minfo_buf_ridx.consumeTail();
                ShouldReturn := TRUE;
            END_IF;

            IF ShouldReturn = TRUE AND CommandId <> 0 THEN
                ResponsePacketPointer^.ele_count := ResponsePacketPointer^.ele_count + 2;
                ResponsePacketPointer^.whead := MessagePackerFb.PackString(pStart := ResponsePacketPointer^.whead, psValue := ADR('id'));
                ResponsePacketPointer^.whead := MessagePackerFb.PackDINT(pStart := ResponsePacketPointer^.whead, diValue := CommandId);

                ResponsePacketPointer^.whead := MessagePackerFb.PackString(pStart := ResponsePacketPointer^.whead, psValue := ADR('ack'));
                ResponsePacketPointer^.whead := MessagePackerFb.PackBool(pStart := ResponsePacketPointer^.whead, bValue := CommandAck);

                MsgPakInfoWrapup(ResponsePacketPointer^);
                GVL.reMP_info_ridx.pushHead();
            END_IF;
        END_IF;
    END_IF;

// --- Reel motor cyclic driver ---
// Two FB instances so we can have one move active while another is
// queued in the axis buffer. SoftMotion rejects >1 movement per FB
// (SMC_MORE_THAN_ONE_MOVEMENT_PER_INSTANCE) so we dispatch to whichever
// FB is idle. BufferMode = Buffered: queued move starts when the active
// one finishes.
IF TRUE THEN
    reelMoveRelative(
        Axis         := reelpullmotor,
        Execute      := reelGoRequest,
        Distance     := reelGoDistance,
        Velocity     := reelGoVelocity,
        Acceleration := reelGoAccel,
        Deceleration := reelGoDecel,
        Jerk         := reelGoJerk,
        BufferMode   := MC_BUFFER_MODE.BlendingHigh
    );
    reelMoveRelative2(
        Axis         := reelpullmotor,
        Execute      := reelGoRequest2,
        Distance     := reelGoDistance,
        Velocity     := reelGoVelocity,
        Acceleration := reelGoAccel,
        Deceleration := reelGoDecel,
        Jerk         := reelGoJerk,
        BufferMode   := MC_BUFFER_MODE.BlendingHigh
    );

    // One-shot: clear both request flags every scan so each new 'ReelGo'
    // produces a fresh rising edge on whichever FB was selected.
    IF reelGoRequest  THEN reelGoRequest  := FALSE; END_IF
    IF reelGoRequest2 THEN reelGoRequest2 := FALSE; END_IF
END_IF;

(* ---- EthercatPOU.st ---- *)
PROGRAM EthercatPOU

VAR CONSTANT
	MOVEMENT_BUFFER_SIZE:UDINT:=50;
END_VAR
VAR
    i               : INT;

	SRGapCounter:INT;
	OUTPUT_Y00:BOOL;
	OUTPUT_Y01:BOOL;
	OUTPUT_Y02:BOOL;

	INPUT_X00:BOOL;
	INPUT_X01:BOOL;
	INPUT_X02:BOOL;

	Axis_PosRead_FB :  ARRAY[0..3] OF MC_ReadActualPosition;

	Axis_Homing_FB :  ARRAY[0..3] OF SM3_Basic.SMC_Homing;

	OUTPUT_MotPos0:DINT;
	INPUT_MotHome0:BOOL;

	OUTPUT_MotPos1:DINT;
	OUTPUT_MotPos2:DINT;
	OUTPUT_MotPos3:DINT;

	pre_MotPos0:DINT;

	HOMEOFFSET_MotPos0:DINT;
	OUTPUT_ResetPos0:BOOL:=FALSE;
	OUTPUT_ResetPos1:BOOL:=FALSE;
	OUTPUT_ResetPos2:BOOL:=FALSE;
	OUTPUT_ResetPos3:BOOL:=FALSE;

	motor_err_rst:BOOL:=TRUE;
	motor_en:BOOL:=TRUE;
	OnBtn_MotErrRst:BOOL;
	OnRunBtnTrigger:BOOL;
	index:INT:=0;

	AxisMult:DINT:=10000;

	AxisTestPulseCount:DINT:=100;

	MoveLinearAbsolute_0: SM3_Robotics.MC_MoveLinearAbsolute;
	//SetBuffer: SMC_SetMovementQueueBuffer;

    MovementBuffer: ARRAY[0..MOVEMENT_BUFFER_SIZE-1] OF SMC_Movement;  // 16 movements buffer

	motionPose:SM3_Robotics.SMC_POS_REF :=( c := (x := 60.0, y := 0.0, z := 0.0, a := 0.0));
	tmp_ptr:POINTER TO BYTE;
	cmd_type:STRING;
	fb_MsgUnPak : FB_MpUnpacker;
	TransitionParameter:ARRAY [0..1]OF LREAL:=[7,0];
	wait:ton;

	MOTION_ERR:BOOL;
	MOTION_ERR_ID:INT;
	MovementId:SMC_Movement_Id;
	latest_ACC_MovementId:SMC_Movement_Id;

	MG_State:INT;

	MC_GroupReadStatus_0: SM3_Robotics.MC_GroupReadStatus;
	ActiveMovementId:SMC_Movement_Id;
	preActiveMovementId:SMC_Movement_Id;

	retryMCMDCD:INT:=0;

	moid_matcher_buf: ARRAY [0..15] OF SMC_Movement_Id;
	moid_matcher_ridx:FB_RingBufferIndex(16);

	readMovementId:SMC_Movement_Id;
	MsgPakQSize:UDINT:=0;

	RunSpeed:REAL:=300;
	RunFactor:REAL:=1;

	DO_HOMING:BOOL:=FALSE;
	HOMING_SENSOR:BOOL:=FALSE;

	HOMING_INDEX:BOOL;
	HOMING_DONE:BOOL;
	HOMING_BUSY:BOOL;

	MotPosIntegral0:DINT:=0;
	IOGapCounter:DINT:=0;
END_VAR

(* =========== IMPLEMENTATION =========== *)
i:=i+1;

IF (i AND 63)=0 THEN
	OUTPUT_Y00:=NOT OUTPUT_Y00;
	SRGapCounter:=0;
END_IF

OUTPUT_Y01:=INPUT_X00;

IF(OUTPUT_Y00<>INPUT_X00)THEN
	SRGapCounter:=SRGapCounter+1;
END_IF

//Application.EthercatPOU.OUTPUT_Y00

MC_GroupReadStatus_0(
	AxisGroup          := AxisGroupGVL_agSpiderR.SpiderR,
	Enable             := 1,
	ActiveMovementId =>ActiveMovementId

	);

MoveLinearAbsolute_0(
	AxisGroup          := AxisGroupGVL_agSpiderR.SpiderR,
	Execute            := 0);

MG_State:=AxisGroupGVL_agSpiderR.SpiderR.m_state;

IF(retryMCMDCD>0)THEN retryMCMDCD:=retryMCMDCD-1; END_IF
MsgPakQSize:=GVL.minfo_buf_ridx.size();
IF(retryMCMDCD=0 AND GVL.minfo_buf_ridx.size()>0 AND moid_matcher_ridx.size()<7)THEN
	tmp_ptr:=ADR(GVL.minfo_buf[GVL.minfo_buf_ridx.getTail()][0]);
	fb_MsgUnPak.Init(ADR(tmp_ptr[1]),tmp_ptr[0]);

	cmd_type:=fb_MsgUnPak.TryReadString('cmd','');

	IF(cmd_type='G1')THEN
		motionPose.c.X:=fb_MsgUnPak.TryReadREAL('X',motionPose.c.X);
		motionPose.c.Y:=fb_MsgUnPak.TryReadREAL('Y',motionPose.c.Y);
		motionPose.c.Z:=fb_MsgUnPak.TryReadREAL('Z',motionPose.c.Z);
		motionPose.c.A:=fb_MsgUnPak.TryReadREAL('A',motionPose.c.A);

		MoveLinearAbsolute_0(
		AxisGroup          := AxisGroupGVL_agSpiderR.SpiderR,
		Execute            := 1,
		Position           := motionPose,              // ← [0.0,0.0,0.0,0.0]
		Velocity           := RunSpeed*3,                 // 速度 (mm/s 或 deg/s)
		Acceleration       := RunSpeed,                // 加速度 (mm/s² 或 deg/s²)
		Deceleration       := RunSpeed,
		Jerk               := RunSpeed/3,
		CoordSystem		   := SMC_COORD_SYSTEM.MCS,

		BufferMode         := SM3_Common.MC_BUFFER_MODE.BlendingHigh, // 緩衝模式
		TransitionMode     := SM3_Robotics.MC_TRANSITION_MODE.TMCornerDistance,
        TransitionParameter:= TransitionParameter,

		//BufferMode         := SM3_Common.MC_BUFFER_MODE.Buffered,
		//TransitionMode     := SM3_Robotics.MC_TRANSITION_MODE.TMNone,

		VelFactor:=RunFactor,
		AccFactor:=RunFactor,
		JerkFactor:=RunFactor,
		TorqueFactor:=1,
		Done=>,
		Busy=>,
		Active=>,
		Error=>MOTION_ERR,
		ErrorID=>MOTION_ERR_ID,
		MovementId=>MovementId
		);

		IF(MoveLinearAbsolute_0.CommandAccepted)THEN
	    	GVL.minfo_buf_ridx.consumeTail();
			latest_ACC_MovementId:=MovementId;

			moid_matcher_buf[moid_matcher_ridx.getHead()]:=latest_ACC_MovementId;
			moid_matcher_ridx.pushHead();
		ELSE
			retryMCMDCD:=50;
		END_IF

	ELSE
	    GVL.minfo_buf_ridx.consumeTail();
	END_IF

END_IF

IF(ActiveMovementId<>0 AND preActiveMovementId<>ActiveMovementId)THEN
	readMovementId:=moid_matcher_buf[moid_matcher_ridx.getTail()];
	moid_matcher_ridx.consumeTail();
END_IF

preActiveMovementId:=ActiveMovementId;

(* ---- POU_BUFFER_RUN.st ---- *)
PROGRAM POU_BUFFER_RUN
VAR CONSTANT
	MOVEMENT_BUFFER_SIZE:UDINT:=50;
END_VAR
VAR
	Axis_PosRead_FB :  ARRAY[0..3] OF MC_ReadActualPosition;

	Axis_Homing_FB :  ARRAY[0..3] OF SM3_Basic.SMC_Homing;

    i               : INT;
	OUTPUT_MotPos0:DINT;
	INPUT_MotHome0:BOOL;
	OUTPUT_Y00:BOOL;
	OUTPUT_Y01:BOOL;
	OUTPUT_Y02:BOOL;

	OUTPUT_MotPos1:DINT;
	OUTPUT_MotPos2:DINT;
	OUTPUT_MotPos3:DINT;

	pre_MotPos0:DINT;

	HOMEOFFSET_MotPos0:DINT;
	OUTPUT_ResetPos0:BOOL:=FALSE;
	OUTPUT_ResetPos1:BOOL:=FALSE;
	OUTPUT_ResetPos2:BOOL:=FALSE;
	OUTPUT_ResetPos3:BOOL:=FALSE;

	motor_err_rst:BOOL:=TRUE;
	motor_en:BOOL:=TRUE;
	OnBtn_MotErrRst:BOOL;
	OnRunBtnTrigger:BOOL;
	index:INT:=0;

	AxisMult:DINT:=10000;

	AxisTestPulseCount:DINT:=100;

	MoveLinearAbsolute_0: SM3_Robotics.MC_MoveLinearAbsolute;
	Waypoints : ARRAY[0..3] OF SM3_Robotics.SMC_POS_REF :=
    [
        ( c := (x := 60.0, y := 0.0, z := 0.0, a := 0.0)),  // Waypoint 0
        ( c := (x := 0.0, y := 60.0, z := 0.0, a := 90.0)), // Waypoint 1
        ( c := (x := -60.0, y := -60.0, z := 0.0, a := 0.0)),  // Waypoint 2
        ( c := (x := 0.0, y := 0.0, z := 0.0, a := 0.0))  // Waypoint 2

    ];
	SetBuffer: SMC_SetMovementQueueBuffer;

    MovementBuffer: ARRAY[0..MOVEMENT_BUFFER_SIZE-1] OF SMC_Movement;  // 16 movements buffer

	motionPose:SM3_Robotics.SMC_POS_REF :=( c := (x := 60.0, y := 0.0, z := 0.0, a := 0.0));
	tmp_ptr:POINTER TO BYTE;
	cmd_type:STRING;
	fb_MsgUnPak : FB_MpUnpacker;
	TransitionParameter:ARRAY [0..1]OF LREAL:=[7,0];
	wait:ton;

	MOTION_ERR:BOOL;
	MOTION_ERR_ID:INT;
	MovementId:SMC_Movement_Id;
	latest_ACC_MovementId:SMC_Movement_Id;

	MG_State:INT;

	MC_GroupReadStatus_0: SM3_Robotics.MC_GroupReadStatus;
	ActiveMovementId:SMC_Movement_Id;
	preActiveMovementId:SMC_Movement_Id;

	retryMCMDCD:INT:=0;

	moid_matcher_buf: ARRAY [0..65] OF SMC_Movement_Id;
	moid_matcher_ridx:FB_RingBufferIndex(66);
	readMovementId:SMC_Movement_Id;
	MsgPakQSize:UDINT:=0;

	RunSpeed:REAL:=300;
	RunFactor:REAL:=1;

	DO_HOMING:BOOL:=FALSE;
	HOMING_SENSOR:BOOL:=FALSE;

	HOMING_INDEX:BOOL;
	HOMING_DONE:BOOL;
	HOMING_BUSY:BOOL;

	MotPosIntegral0:DINT:=0;
	IOGapCounter:DINT:=0;
END_VAR
(* =========== IMPLEMENTATION =========== *)

//OUTPUT_Y00:=OUTPUT_Y00;
motor_en:=TRUE;

motor_err_rst:=OnBtn_MotErrRst;
Axis_PosRead_FB[0](
	Enable := TRUE,
	Axis := IoConfig_Globals.Axis0,
	Valid => ,
	Error => ,
	ErrorID => ,
	Position =>
);

Axis_PosRead_FB[1](
	Enable := TRUE,
	Axis := IoConfig_Globals.Axis1,
	Valid => ,
	Error => ,
	ErrorID => ,
	Position =>
);

Axis_PosRead_FB[2](
	Enable := TRUE,
	Axis := IoConfig_Globals.Axis2,
	Valid => ,
	Error => ,
	ErrorID => ,
	Position =>
);

//OUTPUT_MotPos0:= LREAL_TO_DINT(Axis_PosRead_FB[0].Position/360*AxisMult)+HOMEOFFSET_MotPos0;
//OUTPUT_MotPos1:= LREAL_TO_DINT(Axis_PosRead_FB[1].Position/360*AxisMult);
//OUTPUT_MotPos2:= LREAL_TO_DINT(Axis_PosRead_FB[2].Position/360*AxisMult);

//OUTPUT_MotPos3:= LREAL_TO_DINT(Axis_PosRead_FB[3].Position/360*AxisMult);

(*
IF Axis_PosRead_REAL[3]=0 THEN
	OUTPUT_MotPos3:=0;
ELSE
	OUTPUT_MotPos3:=OUTPUT_MotPos3+AxisTestPulseCount;
END_IF*)

OUTPUT_Y00:=MotPosIntegral0>-100;

Axis_Homing_FB[0](
Axis:=IoConfig_Globals.Axis0,
bExecute:=DO_HOMING,
//fSignalDelay:=0,
fHomePosition:=0,
fVelocityFast:=5,
fVelocitySlow:=1,
fAcceleration:=15,
fDeceleration:=15,
fJerk:=1,
bReturnToZero:=TRUE,
nDirection:=SM3_Basic.MC_DIRECTION.negative,
bReferenceSwitch:=INPUT_MotHome0,//HOMING_SENSOR,//NOT INPUT_MotHome0,
nHomingMode:=SM3_Basic.SMC_HOMING_MODE.FAST_BSLOW_STOP_S,
bIndexOccured:=HOMING_INDEX,

bIgnoreHWLimit:=TRUE,
bDone=>HOMING_DONE,
bBusy=>HOMING_BUSY

);

IF HOMING_DONE THEN
	OUTPUT_ResetPos0:=TRUE;
	OUTPUT_MotPos0:=0;
	pre_MotPos0:=0;

	DO_HOMING:=FALSE;
ELSE
	OUTPUT_ResetPos0:=FALSE;
	MotPosIntegral0:=MotPosIntegral0+OUTPUT_MotPos0-pre_MotPos0;
	//OUTPUT_ResetPos0:=FALSE;
	pre_MotPos0:=OUTPUT_MotPos0;
END_IF

HOMEOFFSET_MotPos0:=0;

//OUTPUT_Y00:=(IOGapCounter AND (1024-1))<2;
IF INPUT_MotHome0 THEN

   OUTPUT_MotPos3:=OUTPUT_MotPos3+10;
END_IF
OUTPUT_Y01:=INPUT_MotHome0;

OUTPUT_Y02:=INPUT_MotHome0;

IOGapCounter:=IOGapCounter+1;

MoveLinearAbsolute_0(
AxisGroup          := AxisGroupGVL_agSpiderR.SpiderR,
Execute            := 0);
MG_State:=AxisGroupGVL_agSpiderR.SpiderR.m_state;

IF(retryMCMDCD>0)THEN retryMCMDCD:=retryMCMDCD-1; END_IF
MsgPakQSize:=GVL.minfo_buf_ridx.size();
IF(retryMCMDCD=0 AND GVL.minfo_buf_ridx.size()>0 AND moid_matcher_ridx.size()<7)THEN
	tmp_ptr:=ADR(GVL.minfo_buf[GVL.minfo_buf_ridx.getTail()][0]);
	fb_MsgUnPak.Init(ADR(tmp_ptr[1]),tmp_ptr[0]);

	cmd_type:=fb_MsgUnPak.TryReadString('cmd','');

	IF(cmd_type='G1')THEN
		motionPose.c.X:=fb_MsgUnPak.TryReadREAL('X',motionPose.c.X);
		motionPose.c.Y:=fb_MsgUnPak.TryReadREAL('Y',motionPose.c.Y);
		motionPose.c.Z:=fb_MsgUnPak.TryReadREAL('Z',motionPose.c.Z);
		motionPose.c.A:=fb_MsgUnPak.TryReadREAL('A',motionPose.c.A);

		MoveLinearAbsolute_0(
		AxisGroup          := AxisGroupGVL_agSpiderR.SpiderR,
		Execute            := 1,
		Position           := motionPose,              // ← [0.0,0.0,0.0,0.0]
		Velocity           := RunSpeed*3,                 // 速度 (mm/s 或 deg/s)
		Acceleration       := RunSpeed,                // 加速度 (mm/s² 或 deg/s²)
		Deceleration       := RunSpeed,
		Jerk               := RunSpeed/3,
		CoordSystem		   := SMC_COORD_SYSTEM.MCS,

		BufferMode         := SM3_Common.MC_BUFFER_MODE.BlendingHigh, // 緩衝模式
		TransitionMode     := SM3_Robotics.MC_TRANSITION_MODE.TMCornerDistance,
        TransitionParameter:= TransitionParameter,

		//BufferMode         := SM3_Common.MC_BUFFER_MODE.Buffered,
		//TransitionMode     := SM3_Robotics.MC_TRANSITION_MODE.TMNone,

		VelFactor:=RunFactor,
		AccFactor:=RunFactor,
		JerkFactor:=RunFactor,
		TorqueFactor:=1,
		Done=>,
		Busy=>,
		Active=>,
		Error=>MOTION_ERR,
		ErrorID=>MOTION_ERR_ID,
		MovementId=>MovementId
		);

		IF(MoveLinearAbsolute_0.CommandAccepted)THEN
	    	GVL.minfo_buf_ridx.consumeTail();
			latest_ACC_MovementId:=MovementId;

			moid_matcher_buf[moid_matcher_ridx.getHead()]:=latest_ACC_MovementId;
			moid_matcher_ridx.pushHead();
		ELSE
			retryMCMDCD:=50;
		END_IF

	ELSE
	    GVL.minfo_buf_ridx.consumeTail();
	END_IF

END_IF

MC_GroupReadStatus_0(
	AxisGroup          := AxisGroupGVL_agSpiderR.SpiderR,
	Enable            := 1,
	ActiveMovementId =>ActiveMovementId

	);

IF(ActiveMovementId<>0 AND preActiveMovementId<>ActiveMovementId)THEN
	readMovementId:=moid_matcher_buf[moid_matcher_ridx.getTail()];
	moid_matcher_ridx.consumeTail();
END_IF

preActiveMovementId:=ActiveMovementId;

(* ---- TCP_MSGPAK_Server.st ---- *)
PROGRAM TCP_MSGPAK_Server
VAR
    CpH : __XWORD;    // Comm task profile: this task's handle
    CpR : UDINT;
    CpP : POINTER TO CmpIecTask.Task_Info2;
    CpOut : LREAL;
    // --- Server Configuration ---
    //
    // Bind to 0.0.0.0 (any interface). Pre-fix the server was bound to a
    // specific machine IP (192.168.1.70); when the PLC ran on a host whose
    // interfaces didn't include that IP, NBS silently failed to listen
    // while still reporting xServerActive=TRUE -- the symptom was raw
    // socket connect refused even though the FSM looked healthy and
    // UiPingCount/AxisGroupSMScans kept climbing. 0.0.0.0 makes the bind
    // succeed on whatever interface the host has, and the OS routes by
    // destination IP from the client side. If a specific-IP bind is ever
    // needed (e.g. firewall pinning), change the literal here -- it's
    // exposed as a GET_DIAG field too (see DrainHostPackets.st).
    //
    // Port: 8125, single-client TCP. See memory ui_plc_single_client_arbitration.
    bEnableServer         : BOOL := TRUE;
    ipServerAddress       : NBS.IPv4Address := (ipAddress:='0.0.0.0');
    uiServerPort          : UINT := 8125;

    // --- The Server Function Block Instance ---
    fbMyServer            : FB_TcpMsgPakServer;

    // --- Logic for Packet Flow Control ---
    REEN_CD               : INT := 0;

    recv_counter          : INT := 0;
    TMP_PKT_IDX           : UDINT := 0;

	tmp_MsgPakInfo_ptr:POINTER TO MsgPakInfo;
	tmp_ptr:POINTER TO BYTE;

	// Send-stall recovery: if Send() keeps returning FALSE while the
	// socket reports xActive=TRUE (half-open / TX backpressure), the
	// reply ring would fill up forever. Drop the head packet after
	// SEND_MAX_RETRIES consecutive cycles and count it. See
	// doc/3-subsystems/ringbuf-bugs.md #7.
	send_retry_count: UDINT := 0;
	// A reply that cannot be sent for SEND_STALL_TIME is dropped. Keeps the
	// ring from filling up behind one stuck packet during a half-open TX
	// stall (xActive=TRUE but Send returns FALSE). See ringbuf-bugs.md #7.
	// It was 20 Comm scans (100 ms at 5 ms); a timer keeps it 100 ms
	// whatever the Comm period (1 ms since 2026-09-25).
	SEND_STALL_TIME: TIME := T#100MS;
	sendStallTimer: Standard.TON;

	// TX-side half-open escalation: count consecutive head-drops with no
	// successful Send between them. After the threshold, signal
	// FB_TcpMsgPakServer to force a socket reset so a fresh client can
	// reconnect. Reset to 0 on any successful Send. 5 head-drops at
	// ~100ms apart -> ~500ms of sustained TX stall before reclaiming
	// the socket; well under any human-perceivable hang and far above
	// transient TCP backpressure.
	consecutive_stall_drops: UDINT := 0;
	TX_STALL_DROP_THRESHOLD: UDINT := 5;
	tx_stall_force_reset: BOOL := FALSE;

	DBG_reMP_info_ridx_size:INT;

	// Routing of inbound packets (GVL minfo_buf / sysinfo_buf).
	RouteUnpacker : FB_MpUnpacker;
	RouteType     : STRING;
	RouteCmd      : STRING;
	RouteToSys    : BOOL;
	CommIter      : INT;     // packets taken / replies sent this scan
END_VAR
(* =========== IMPLEMENTATION =========== *)
// Comm task profile (GVL.Comm*): last scan's task time vs its POU span
CpH := CmpIecTask.IecTaskGetCurrent(ADR(CpR));
IF CpR = 0 THEN
    CpP := CmpIecTask.IecTaskGetInfo3(CpH, ADR(CpR));
    IF (CpR = 0) AND (CpP <> 0) THEN
        CpOut := DWORD_TO_LREAL(CpP^.dwCycleTime) - GVL.CommScanUsLast;
        GVL.CommTaskUsMax := MAX(GVL.CommTaskUsMax, DWORD_TO_LREAL(CpP^.dwCycleTime));
        GVL.CommOutsideUsMax := MAX(GVL.CommOutsideUsMax, CpOut);
        IF CpOut > 500.0 THEN
            GVL.CommOutsideOver500 := GVL.CommOutsideOver500 + 1;
        END_IF;
    END_IF;
END_IF;
GVL.CommT[0] := LTIME(); GVL.CommCyc[0] := GVL.EcProfCycles;   // Comm task profile (GVL.Comm*)

//==================================================================================================
// PROGRAM IMPLEMENTATION
//==================================================================================================

IF REEN_CD>0 THEN
	REEN_CD:=REEN_CD-1;
END_IF

// --- 4. Call the server function block instance ---
// The PKT_ALLOW_NEXT input is now controlled by our logic.
// Up to GVL.CommPacketsPerScan packets per scan: the FB exposes one packet
// per call, so it is called again while the last call produced one and
// both rings still have room. Bytes already in its buffer need no new read.
FOR CommIter := 1 TO MAX(1, GVL.CommPacketsPerScan) DO
fbMyServer(
    ENABLE:= bEnableServer,
    IP_ADDRESS:= ipServerAddress,
    PORT:= uiServerPort,
    PKT_ALLOW_NEXT:=(GVL.minfo_buf_ridx.Space()>1) AND (GVL.sysinfo_buf_ridx.Space()>1),
    xForceReset:= tx_stall_force_reset
);
// One-shot pulse: clear after delivery so we don't loop-reset.
tx_stall_force_reset := FALSE;

// This IF statement will be TRUE for one cycle when a new packet arrives.
IF fbMyServer.PKT_IDX > TMP_PKT_IDX THEN
	REEN_CD:=50;
    recv_counter := recv_counter + 1;
	GVL.HostRxCount := GVL.HostRxCount + 1;

	// Length guard: slots are 256 bytes (1 len + 255 payload). Over-length
	// packets would wrap via DINT_TO_BYTE and corrupt the slot silently.
	// See doc/3-subsystems/ringbuf-bugs.md #1. Type/cmd dispatch happens in AxisGroupSM
	// after the slot is drained; unrecognised types NAK with
	// 'missing_type_field'.
	IF (fbMyServer.BUFFER_LEN > GVL.MAX_SLOT_PAYLOAD) THEN
		GVL.OverlenDropCount := GVL.OverlenDropCount + 1;
		// It used to vanish without a reply, leaving the host to time out.
		IF NOT GVL.OverlenNakPending THEN
			RouteUnpacker.Init(ADR(fbMyServer.BUFFER_PTR[0]), DINT_TO_UDINT(fbMyServer.BUFFER_LEN));
			GVL.OverlenNakId := TO_DINT(RouteUnpacker.TryReadINT64('id', 0));
			GVL.OverlenNakPending := GVL.OverlenNakId <> 0;
		END_IF;
	ELSE
		// Order-free SYS commands take their own ring so they never queue
		// behind a motion packet the PLC cannot take yet. Everything else
		// -- motion, and SYS whose order against motion matters
		// (COORD1_BIND/UNBIND, SCRATCHPAD_WRITE, unknown) -- stays FIFO in
		// minfo_buf. Unparseable packets go to minfo_buf too, where the
		// drain loop NAKs them as before.
		RouteUnpacker.Init(ADR(fbMyServer.BUFFER_PTR[0]), DINT_TO_UDINT(fbMyServer.BUFFER_LEN));
		RouteType := RouteUnpacker.TryReadString('type', '');
		RouteCmd  := RouteUnpacker.TryReadString('cmd', '');
		RouteToSys := (RouteType = 'SYS') AND (
			RouteCmd = 'PING' OR RouteCmd = 'GA_EV' OR RouteCmd = 'GET_MACHINE_STATE'
			OR RouteCmd = 'GET_DIAG' OR RouteCmd = 'VERSION' OR RouteCmd = 'RESET_DBG_INFO'
			OR RouteCmd = 'SET_AXIS_SIM' OR RouteCmd = 'GET_COORD1_DEBUG' OR RouteCmd = 'EVT_MARK'
			OR RouteCmd = 'PLAN_GET' OR RouteCmd = 'SET_OVERRIDE' OR RouteCmd = 'DI_WATCH' OR RouteCmd = 'TASK_STATS'
			OR RouteCmd = 'AXIS_INFO' OR RouteCmd = 'IO_STATE' OR RouteCmd = 'EC_STATS'
			OR RouteCmd = 'JOINT_MOVE' OR RouteCmd = 'JOINT_STOP' OR RouteCmd = 'JOINT_STATE');
		IF RouteToSys AND (GVL.sysinfo_buf_ridx.Space() > 0) THEN
			tmp_ptr:=ADR(GVL.sysinfo_buf[GVL.sysinfo_buf_ridx.GetHead()][0]);
			tmp_ptr[0]:=DINT_TO_BYTE(fbMyServer.BUFFER_LEN);
			MEMUtils.MemCpy(ADR(tmp_ptr[1]),ADR(fbMyServer.BUFFER_PTR[0]),DINT_TO_UINT(fbMyServer.BUFFER_LEN));
			GVL.sysinfo_buf_ridx.PushHead();
		ELSIF (NOT RouteToSys) AND (GVL.minfo_buf_ridx.Space() > 0) THEN
			tmp_ptr:=ADR(GVL.minfo_buf[GVL.minfo_buf_ridx.GetHead()][0]);
			tmp_ptr[0]:=DINT_TO_BYTE(fbMyServer.BUFFER_LEN);
			MEMUtils.MemCpy(ADR(tmp_ptr[1]),ADR(fbMyServer.BUFFER_PTR[0]),DINT_TO_UINT(fbMyServer.BUFFER_LEN));
			GVL.minfo_buf_ridx.PushHead();
		END_IF;
	END_IF;
END_IF;

// Update the packet index tracker
IF fbMyServer.PKT_IDX = TMP_PKT_IDX THEN
	EXIT;                  // no packet this call: nothing more buffered
END_IF;
TMP_PKT_IDX := fbMyServer.PKT_IDX;
END_FOR;

DBG_reMP_info_ridx_size:=GVL.reMP_info_ridx.Size();
// Up to GVL.CommPacketsPerScan replies per scan (acks, events, MOVE_DONE,
// heartbeat all queue here); stop at the first one that cannot be sent.
FOR CommIter := 1 TO MAX(1, GVL.CommPacketsPerScan) DO
IF GVL.reMP_info_ridx.Size() = 0 THEN
	EXIT;
END_IF;
IF GVL.reMP_info_ridx.Size()>0 THEN
	IF fbMyServer.xResetting OR NOT fbMyServer.CLIENT.xActive THEN
		// Socket is dying (reset in flight) or already dead. Continuing
		// to Send would either succeed-then-lose-the-reply (client gone,
		// ConsumeTail already ran) or fail and pump the stall counter
		// for no reason. Flush the backlog so we don't replay stale
		// replies to whatever client connects next.
		WHILE GVL.reMP_info_ridx.Size() > 0 DO
			GVL.reMP_info_ridx.ConsumeTail();
		END_WHILE;
		send_retry_count := 0;
		sendStallTimer(IN := FALSE);
		consecutive_stall_drops := 0;
	ELSE
		tmp_MsgPakInfo_ptr:=ADR(GVL.reMP_info_arr[GVL.reMP_info_ridx.GetTail()]);
		// Only consume the slot if the TCP write succeeded. A transient
		// failure (xActive=TRUE, Send=FALSE) means TX-side backpressure;
		// leave the packet so it retries next cycle or escalates below.
		IF fbMyServer.Send(BUFFER_PTR := tmp_MsgPakInfo_ptr^.buf, BUFFER_LEN := tmp_MsgPakInfo_ptr^.buf_size) THEN
			GVL.reMP_info_ridx.ConsumeTail();
			send_retry_count := 0;
			sendStallTimer(IN := FALSE);
			// Successful Send proves the TX path is alive; clear the
			// half-open escalation counter.
			consecutive_stall_drops := 0;
		ELSE
			// xActive=TRUE but Send returned FALSE -> TX stall / half-open.
			// (Hard Write errors now raise xResetConnection inside Send.st,
			// so by next cycle xResetting will be TRUE and we'll hit the
			// flush branch above; the stall escalation here only fires on
			// pure backpressure where Write reported NO_ERROR but the
			// socket isn't draining.) See doc/3-subsystems/ringbuf-bugs.md #7.
			send_retry_count := send_retry_count + 1;
			sendStallTimer(IN := TRUE, PT := SEND_STALL_TIME);
			IF sendStallTimer.Q THEN
				GVL.reMP_info_ridx.ConsumeTail();
				GVL.SendStallDropCount := GVL.SendStallDropCount + 1;
				send_retry_count := 0;
				sendStallTimer(IN := FALSE);
				// TX-side half-open escalation. Each head-drop = ~100ms of
				// stall. Once we accumulate TX_STALL_DROP_THRESHOLD in a
				// row, the socket is genuinely dead from our side; raise
				// xForceReset so the FB tears down the connection and a
				// new client can reconnect.
				consecutive_stall_drops := consecutive_stall_drops + 1;
				IF consecutive_stall_drops >= TX_STALL_DROP_THRESHOLD THEN
					tx_stall_force_reset := TRUE;
					consecutive_stall_drops := 0;
				END_IF;
			END_IF;
			EXIT;              // TX not draining: try again next scan
		END_IF;
	END_IF;
END_IF
END_FOR;

// --- MsgPack self-test harness hook (Comm task; runs cyclically).
// See doc/2-contracts/msgpack.md and FB_MsgPackTests. Toggle GVL.bRunMsgPackTests
// in online mode to fire; results on GVL.fbMsgPackTests.*.
GVL.fbMsgPackTests(bRun := GVL.bRunMsgPackTests);

(* ---- TCP_Server.st ---- *)
PROGRAM TCP_Server
VAR CONSTANT
    // --- Define the maximum size of the incoming and outgoing data ---
    mySize : UDINT := 1024;

    // --- Prefix to add to incoming data as a BYTE array (currently unused in echo logic) ---
    // ASCII values for "echo:" (e=16#65, c=16#63, h=16#68, o=16#6F, :=16#3A)
    //cEchoPrefix : ARRAY [0..4] OF BYTE := [16#65, 16#63, 16#68, 16#6F, 16#3A];
    LEN_ECHO_PREFIX : UDINT := 5; // Length of the "echo:" prefix

    // --- String "HR" to send periodically ---
    cHRString : ARRAY [0..1] OF BYTE := [16#48, 16#52]; // ASCII for "HR"
    LEN_HR_STRING : UDINT := 2; // Length of "HR"
END_VAR

VAR
    // --- Server and Connection Function Blocks ---
    myIPAddress : NBS.IPv4Address := (ipAddress:='192.168.3.6');
    myServer : NBS.TCP_Server := (
        itfIPAddress:=myIPAddress,
        uiPort:=8123,
		xEnable:=TRUE,
		udiMaxConnections:=1
    );
    itfServer : NBS.IServer;
    xServerActive : BOOL;

    myConnection : NBS.TCP_Connection;
    xEnableConnection : BOOL; // Controls the actual enable input of myConnection

    // --- Data Buffers and Counters ---
    udiBytesReceived : UDINT;
    eReadErrorID, eWriteErrorID : NBS.ERROR;
    sSendBuffer : ARRAY [0..mySize + LEN_ECHO_PREFIX - 1] OF BYTE; // BYTE array for outgoing data (sized for prefix + data)
    udiBytesToSend : UDINT; // Actual number of bytes to send in the current cycle

    // --- State Control for Connection Management ---
    xResetConnection : BOOL := FALSE;      // Flag to initiate a connection reset process
    xLastConnectionActive : BOOL := FALSE; // Holds the state of xActive from the previous cycle

    // --- Delay Timer for Connection Reset ---
    fbResetDelayTimer : Standard.TON;      // TON function block for the delay
    xDelayDone : BOOL;                     // Output of the TON timer

	fb_MsgPakParser : FB_MsgPakLevelParser;

	bufferbuffer: ARRAY [0..1024-1] OF BYTE;
	dbuffer:FB_DataBuffer;
	i : DINT;
	curPacketStartIdx:DINT;
	curPacketLen:DINT;
	TMP_buffer_ptr : POINTER TO BYTE;
	TMP_buff_size:DINT:=0;

	fb_MsgUnPak : FB_MpUnpacker;
	data_type:STRING;
	cmd_type:STRING;
	//motionPose:SM3_Robotics.SMC_POS_REF:= ( c := (x := 00.0, y := 0.0, z := 0.0, a := 0.0));

	tmp_ptr:POINTER TO BYTE;

	INIT:BOOL:=TRUE;

	fbWaitTimeout   : TON;         // Timer to escape the blocking loop

END_VAR
(* =========== IMPLEMENTATION =========== *)

IF INIT THEN
	fb_MsgPakParser.ResetParser();
	dbuffer.reset_buffer(ADR(bufferbuffer[0]),SIZEOF(bufferbuffer));
	INIT:=FALSE;
END_IF
// -----------------------------------------------------------------------------
// MAIN LOGIC
// -----------------------------------------------------------------------------

// 1. Enable and run the TCP server.
myServer();

// Get the server's interface pointer.
itfServer := myServer.itfServer;
xEnableConnection := xServerActive;
xServerActive := itfServer <> 0;

// 2. Control the TCP connection function block's enable input with a delay.

// If a reset is initiated (xResetConnection is TRUE)...
IF xResetConnection THEN
    // Start the delay timer. Its IN is TRUE as long as xResetConnection is TRUE.
    fbResetDelayTimer(IN := TRUE, PT := T#10MS, Q => xDelayDone);

    // If the delay timer is done (Q is TRUE), then disable the connection.
    IF xDelayDone THEN
        xEnableConnection := FALSE;
		fb_MsgPakParser.ResetParser();
		dbuffer.clear();
    END_IF
ELSE
    // If no reset is initiated, ensure the timer is reset.
    fbResetDelayTimer(IN := FALSE);
    xDelayDone := FALSE; // Ensure xDelayDone is false when timer is off
END_IF

// Call the connection block with the controlled enable input.
myConnection(itfServer:=itfServer, xEnable:=xEnableConnection);

// 3. Main communication logic for an active connection.
IF myConnection.xActive THEN

    // --- Read from the client ---
    eReadErrorID := myConnection.Read(
        dbuffer.get_head(), // Address of the first byte in the array
        dbuffer.get_space(), // Total size of the buffer in bytes
        udiCount => udiBytesReceived // Number of bytes actually received
    );
	dbuffer.write_length(udiBytesReceived);

	(*eWriteErrorID := myConnection.Write(
            ADR(sSendBuffer[0]), // Address of the first byte to send
            udiBytesToSend // Number of bytes to send
        );*)

    // Check if data was successfully read without error and if any bytes were received.
    IF eReadErrorID = 0 AND dbuffer.size() > 0 THEN

		curPacketStartIdx:=0;
		curPacketLen:=0;
		TMP_buffer_ptr:=dbuffer.get_buffer();
		TMP_buff_size:=dbuffer.size();
		FOR i := dbuffer.size()-UDINT_TO_DINT(udiBytesReceived) TO dbuffer.size() - 1 DO
			fb_MsgPakParser(in_byte := TMP_buffer_ptr[i]);//feed in latest data
			IF fb_MsgPakParser.e_error = E_MsgPakLevelParser_ERROR.NONE THEN

				IF fb_MsgPakParser.ui_level_stack_size = 0 THEN
					//a packet
					curPacketLen:=i-curPacketStartIdx+1;

					IF(curPacketLen<2) THEN//too short, might be an parse error
						//E_MsgPakLevelParser_ERROR.UNEXPECTED_BYTE;
						xResetConnection:=TRUE;
						EXIT;
					ELSE
						fb_MsgUnPak.Init(ADR(TMP_buffer_ptr[curPacketStartIdx]),curPacketLen);

						data_type:=fb_MsgUnPak.TryReadString('type','');

						IF(data_type='M')THEN//motion type
							WHILE GVL.minfo_buf_ridx.space() = 0 DO//dead wait
								// The timer must be called repeatedly inside the loop to make it run.
								fbWaitTimeout(IN:= TRUE, PT:= UDINT_TO_TIME(1));

								// If the timer's output (Q) becomes TRUE, exit the loop.
								IF fbWaitTimeout.Q THEN
									EXIT; // Exit the WHILE loop immediately
								END_IF;
							END_WHILE

							// space() returns UDINT — was >=0 (always true). Need free slot before writing.
							IF(GVL.minfo_buf_ridx.space() > 0)THEN
								tmp_ptr:=ADR(GVL.minfo_buf[GVL.minfo_buf_ridx.getHead()][0]);
								tmp_ptr[0]:=DINT_TO_BYTE(curPacketLen);//keep data len
								//MEM.MemMove(ADR(TMP_buffer_ptr[curPacketStartIdx]),ADR(tmp_ptr[1]),DINT_TO_UINT(curPacketLen));
								MEMUtils.MemCpy(ADR(tmp_ptr[1]),ADR(TMP_buffer_ptr[curPacketStartIdx]),DINT_TO_UINT(curPacketLen));
								GVL.minfo_buf_ridx.pushHead();
							END_IF

						END_IF

	        			udiBytesToSend := curPacketLen;

						MEMUtils.MemCpy(ADR(sSendBuffer[0]), ADR(TMP_buffer_ptr[curPacketStartIdx]), curPacketLen);
				        eWriteErrorID := myConnection.Write(
				            ADR(sSendBuffer[0]), // Address of the first byte to send
				            udiBytesToSend // Number of bytes to send
				        );
						curPacketStartIdx:=i+1;

					END_IF

				END_IF
			ELSE
				xResetConnection:=TRUE;
				EXIT;

			END_IF
		END_FOR
		IF(curPacketStartIdx<>0) THEN
			dbuffer.move_left(curPacketStartIdx);
		END_IF

		//dbuffer.clear();
    END_IF

END_IF // END IF myConnection.xActive

// 4. Connection tear-down and reset initiation logic.
// This is where a disconnect or error is detected, which then starts the delay.

// A) Detect a graceful disconnect (falling edge of xActive).
IF xLastConnectionActive AND NOT myConnection.xActive THEN
    xResetConnection := TRUE; // Initiate the reset process
END_IF

// B) Detect an abrupt disconnect (error).
IF myConnection.xError THEN
    xResetConnection := TRUE; // Initiate the reset process
END_IF

// C) Complete the reset process.
// Clear the xResetConnection flag ONLY when the delay is over (xDelayDone TRUE)
// AND the connection has actually become inactive (myConnection.xActive FALSE).
IF xResetConnection AND xDelayDone AND NOT myConnection.xActive THEN
    xResetConnection := FALSE; // Reset process is complete
END_IF

// 5. Update the state of the connection for the next PLC cycle.
xLastConnectionActive := myConnection.xActive;

(* ---- TCP_Server_Mult.st ---- *)
PROGRAM TCP_Server_Mult
VAR CONSTANT
    // --- Define the maximum size of the incoming and outgoing strings ---
    mySize : UDINT := 1024;
    // --- Maximum number of simultaneous connections the server will handle ---
    MAX_CONNECTIONS : UINT := 5; // Example: Allow up to 5 concurrent clients
END_VAR

VAR
    // --- Server Function Block ---
    myIPAddress : NBS.IPv4Address := (ipAddress:='192.168.3.6');
    myServer : NBS.TCP_Server := (
        itfIPAddress:=myIPAddress,
        uiPort:=8123,
		xEnable:=TRUE,
		udiMaxConnections:=MAX_CONNECTIONS // Allow multiple connections
    );
    itfServer : NBS.IServer;
    xServerActive : BOOL;

    // --- Array of Connection Function Blocks ---
    myConnections : ARRAY [1..MAX_CONNECTIONS] OF NBS.TCP_Connection;

    // --- Data Buffers and Error IDs (Arrays for each connection) ---
    udiBytesReceived : ARRAY [1..MAX_CONNECTIONS] OF UDINT;
    eReadErrorID : ARRAY [1..MAX_CONNECTIONS] OF NBS.ERROR;
    eWriteErrorID : ARRAY [1..MAX_CONNECTIONS] OF NBS.ERROR;
    sReceiveBuffer : ARRAY [1..MAX_CONNECTIONS] OF STRING(mySize);
    sSendBuffer : ARRAY [1..MAX_CONNECTIONS] OF STRING(mySize + 10); // Prefix + data

    // --- State Control for Connection Management (Arrays for each connection) ---
    xResetConnection : ARRAY [1..MAX_CONNECTIONS] OF BOOL;      // Flag to initiate a reset process for each connection
    xLastConnectionActive : ARRAY [1..MAX_CONNECTIONS] OF BOOL; // Holds the state of xActive from previous cycle for each connection

    // --- Delay Timers for Connection Reset (Arrays for each connection) ---
    fbResetDelayTimer : ARRAY [1..MAX_CONNECTIONS] OF Standard.TON;

    // --- Loop Counter ---
    i : UINT; // Loop variable for iterating through connections
END_VAR
(* =========== IMPLEMENTATION =========== *)

// -----------------------------------------------------------------------------
// MAIN LOGIC
// -----------------------------------------------------------------------------

// 1. Enable and run the TCP server.
myServer();

// Get the server's interface pointer.
itfServer := myServer.itfServer;
xServerActive := itfServer <> 0;

// 2. Loop through each possible connection slot.
FOR i := 1 TO MAX_CONNECTIONS DO

    // --- Control the TCP connection function block's enable input with a delay ---
    // The connection should be enabled by default (when server is active).
    // It's disabled only after the reset delay completes.
    myConnections[i](itfServer:=itfServer, xEnable:=xServerActive AND NOT fbResetDelayTimer[i].Q);

    // 3. Main communication logic for an active connection.
    IF myConnections[i].xActive THEN

        // --- Read from the client ---
        eReadErrorID[i] := myConnections[i].Read(
            ADR(sReceiveBuffer[i]),
            SIZEOF(sReceiveBuffer[i]),
            udiCount => udiBytesReceived[i]
        );

        // Check if data was successfully read without error.
        IF eReadErrorID[i] = 0 AND udiBytesReceived[i] > 0 THEN

            // --- Process the received data ---
            sReceiveBuffer[i][udiBytesReceived[i]] := 0; // Null-terminate the string
            sSendBuffer[i] :=CONCAT(UINT_TO_STRING(i), CONCAT('echo:', sReceiveBuffer[i])); // Add prefix

            // --- Send the echoed data back to the client ---
            eWriteErrorID[i] := myConnections[i].Write(
                ADR(sSendBuffer[i]),
                LEN(sSendBuffer[i])
            );
            sReceiveBuffer[i] := ''; // Clear receive buffer

        END_IF
    END_IF

    // 4. Connection tear-down and reset initiation logic (per connection).
    // This is where a disconnect or error is detected, which then starts the delay for THIS connection.

    // A) Detect a graceful disconnect (falling edge of xActive).
    IF xLastConnectionActive[i] AND NOT myConnections[i].xActive THEN
        xResetConnection[i] := TRUE; // Initiate the reset process for this connection
    END_IF

    // B) Detect an abrupt disconnect (error).
    IF myConnections[i].xError THEN
        xResetConnection[i] := TRUE; // Initiate the reset process for this connection
    END_IF

    // C) Timer Logic for the 100ms delay before actual reset.
    // The timer starts when xResetConnection[i] becomes TRUE.
    fbResetDelayTimer[i](IN := xResetConnection[i], PT := T#100MS);

    // D) Complete the reset process.
    // Clear the xResetConnection[i] flag ONLY when the delay is over (fbResetDelayTimer[i].Q is TRUE)
    // AND the connection has actually become inactive (myConnections[i].xActive is FALSE).
    IF xResetConnection[i] AND fbResetDelayTimer[i].Q AND NOT myConnections[i].xActive THEN
        xResetConnection[i] := FALSE; // Reset process for this connection is complete
    END_IF

    // 5. Update the state of this connection for the next PLC cycle.
    xLastConnectionActive[i] := myConnections[i].xActive;

END_FOR // End of FOR loop

(* ---- WebServer_SIMPLE.st ---- *)
PROGRAM WebServer_SIMPLE
VAR CONSTANT
    mySize : UDINT := 1255;
END_VAR

VAR CONSTANT
    // --- Define your simple HTML page as a constant ---
    sHtmlBody : STRING(1024) :=
        '<!DOCTYPE html><html><head><title>PLC Status</title></head><body><h1>Hello from my CoDeSys PLC!</h1><p>This page is served directly from the controller.</p></body></html>';

    // --- Define the HTTP header template ---
    // We REMOVE the 'Connection: close' header to keep the connection alive.
    // We use a placeholder 'LL' which we will replace with the actual length.
    sHttpHeaderTemplate : STRING(1024) :=
        'HTTP/1.1 200 OK$r$nContent-Type: text/html$r$nContent-Length: LL$r$n$r$n'; // Removed 'Connection: close'
END_VAR

VAR
    /// The certificate of the client should be located in the store under the trusted folder!!

    myIPAddress : NBS.IPv4Address := (ipAddress:='192.168.3.6');
    sMyCommonName : STRING := 'MyPLCserverName';

    myConnection : NBS.TCP_Connection;
    xConnectionReset : BOOL; // Flag to control the connection reset

    myServer : NBS.TCP_Server := (
        itfIPAddress:=myIPAddress,
        uiPort:=8123,
		xEnable:=TRUE,
		udiMaxConnections:=1
    );

    itfServer : NBS.IServer;
    xActive : BOOL;

    udiServerCount : UDINT;
    eServerTxErrorID, eServerRxErrorID : NBS.ERROR;
    myServerData : STRING(mySize);

	sFullHttpResponse : STRING(2024); // Make sure this is large enough
    sContentLength    : STRING(4);    // To hold the string version of the length
END_VAR
(* =========== IMPLEMENTATION =========== *)

// Set myServer.xEnable to start
myServer();

itfServer := myServer.itfServer;
xActive := itfServer <> 0;

// Call the connection block. We control its enable input using a reset flag.
myConnection(itfServer:=itfServer, xEnable:=xActive AND NOT xConnectionReset);

IF myConnection.xActive THEN
    // The connection is active. Read data from the client.
    eServerRxErrorID := myConnection.Read(ADR(myServerData), mySize, udiCount=>udiServerCount);
    IF eServerRxErrorID = 0 AND udiServerCount > 0 THEN
        // A new request was received.

		        // ---- 1. BUILD THE HTTP RESPONSE ----

        // Clear the response string
        sFullHttpResponse := '';

        // Calculate the length of the HTML body and convert it to a string
        sContentLength := DINT_TO_STRING(LEN(sHtmlBody));

        // Build the header by replacing the 'LL' placeholder with the actual length
        sFullHttpResponse := REPLACE(STR1:=sHttpHeaderTemplate, STR2:=sContentLength, L:=LEN(sContentLength), P:=FIND(sHttpHeaderTemplate, 'LL'));

        // Append the HTML body to the headers
        sFullHttpResponse := CONCAT(sFullHttpResponse, sHtmlBody);

        // ---- 2. SEND THE RESPONSE ----
        eServerTxErrorID := myConnection.Write(
                                ADR(sFullHttpResponse),
                                LEN(sFullHttpResponse)
                            );

        // ---- 3. DO NOT CLOSE THE CONNECTION ----
        // The server now waits for the next request on the same connection.
	END_IF
END_IF

// This is the crucial part for tearing down the connection:
// How the PLC detects a client disconnect and resets the connection stack.

// 1. Detect if the connection has an error.
//    This happens on an abrupt disconnect (e.g., pulling the network cable).
IF myConnection.xError THEN
    // An error occurred. Set the reset flag to tear down the connection.
    xConnectionReset := TRUE;
END_IF

// 2. After setting the reset flag, the connection function block needs to be
//    disabled for at least one PLC cycle to reset.
//    Once it's no longer active, we can clear the flag.
IF xConnectionReset AND NOT myConnection.xActive THEN
    // The connection has been torn down. We are ready to accept a new one.
    xConnectionReset := FALSE;
END_IF
